(* IEC 61131-3 sources: BLM_BACKGROUND/src/PROGRAM_FILES/FC (part 3) *)

		GENERAL_STATE#STATE_END:
			CURRENT_STATE:=GENERAL_STATE#STATE_INIT;

	END_CASE;
	OutputState:=CURRENT_STATE;
END_FUNCTION_BLOCK

/*****************************************************************************
 * CHECKS WHETHER THE PIPE IS PRESENT ON THE^AL AND IS READY FOR LOADING, IF *
 *          NEGATIVE IT SETS THE STATUS AND POSITION TO UNDEFINED.           *
 *           IT ALSO RESETS OUTPUTS THAT CONTROL HAZARDOUS DEVICES           *
 *****************************************************************************/

FUNCTION_BLOCK FB_ResetAL

  VAR_EXTERNAL
    i_sys_OPMODE                          : INT;
    i_sys_current_prog	                  :INT;
    i_sys_AL_Robot                        :BOOL;
    OAddress                              : ARRAY [0..MAXDIGITALOUTPUT] OF Digital_Output;
    Disp                                  :ARRAY[(FIRST_DEVICE)..(FIRST_DEVICE+_MAXDEVICES#MAXDEVICES-1)] OF Device;
  END_VAR

  VAR_EXTERNAL CONSTANT
    AUTOMODE                              :INT;
    PROGRAM_JOG                      	    :SINT;
    TIPO_AL42                          	  :SINT;
    TIPO_AL42PLUS                      	  :SINT;
    MAXDIGITALOUTPUT                      :INT;
    OUT_ALZO_SOSTEGNO_TUBO_AL42           :INT;
    OUT_ABBASSO_SOSTEGNO_TUBO_AL42        :INT;
    CLAMP_CARGE                           :INT;
    FIRST_DEVICE                          :INT;
    AL42_STATO_CARICO                  	  :SINT;
    AT_STATE_UNDEFINED                	  :SINT;
    TIPO_AL5                          	  :SINT;
    TIPO_AL5_ROLAND                    	  :SINT;		//AL5 con sistema di misura ROLAND
    TIPO_AL5_LUNGO                    	  :SINT;
    AL5_CARICO_MACCHINA                	  :SINT;	//AL con tubo pronto in posizione di
                                                                //carico tubo in macchina con pinze
                                                                //chiuse, se presente traslatore avanti
    TIPO_AL5_BUNDLE                    	:SINT;
    TIPO_AL5_ROLAND_BUNDLE            	:SINT;		//AL5+BUNDLE con sistema di misura ROLAND
    TIPO_AL5_LUNGO_BUNDLE              	:SINT;	//AL5 speciale lungo 6mt+BUNDLE con sistema di misura ROLAND
    TIPO_MS0017                        	:SINT;	//Caricatore per ditta Sogefi
    TIPO_AL5_FUTABA                    	:SINT;	//Caricatore per ditta Futaba con ricerca saldatura Roland
    OUT_PRESSIONE_PNEUMATICA_AL         :INT;
  END_VAR

  VAR
    dwret     :DWORD;
    TipoAl    :SINT;
    dret      :DINT;
    Address   :DINT;
    StatoAsse :LREAL;
    Programma :INT;

		CURRENT_STATE:INT:=GENERAL_STATE#STATE_INIT;
		AL5_Sollevatore	:FB_AL5_Sollevatore;
		AL5Catene				:FB_AL5Catene;
  END_VAR
	VAR_OUTPUT
		OutputState:INT;
	END_VAR
	CASE CURRENT_STATE OF
		GENERAL_STATE#STATE_INIT:
			IF i_sys_OpMode=AUTOMODE THEN
				Programma:=I_SYS_Current_Prog;
			ELSE
				Programma:=PROGRAM_JOG;
			END_IF;
			// {#ifdef AL_BLM}
				i_sys_AL_Robot:=FALSE;
    		TipoAl:=IndicaTipoAl();
				CASE TipoAL OF
					TIPO_AL42, TIPO_AL42PLUS:
						//Abilitazione forzatura uscite
						oaddress[OUT_ALZO_SOSTEGNO_TUBO_AL42].enable_forzatura:=FALSE;
						oaddress[OUT_ABBASSO_SOSTEGNO_TUBO_AL42].enable_forzatura:=FALSE;
						(*dwret:=_resetTaskId(_task.motiontask_AL);*)
						Disp[CLAMP_CARGE].in_movimento:=FALSE;
						IF TestALReady()=TRUE THEN
							ImpostaAL(Stato:=AL42_STATO_CARICO, Movimento:=FALSE);
						ELSE
							//Stato CARICO AL42 non compatibile con la situazione reale dei
							//dispositivi quindi si mette ad indefinito lo stato del sistema
							Disp[CLAMP_CARGE].stato:=AT_STATE_UNDEFINED;
							Disp[CLAMP_CARGE].position:=AT_STATE_UNDEFINED;
						END_IF;
						CURRENT_STATE:=_FB_ResetAL#STATE_RESET_AL_RESET_USCITE_CARICO;

					TIPO_AL5, TIPO_AL5_ROLAND, TIPO_AL5_LUNGO:
						oaddress[OUT_ALZO_SOSTEGNO_TUBO_AL42].enable_forzatura:=FALSE;
						oaddress[OUT_ABBASSO_SOSTEGNO_TUBO_AL42].enable_forzatura:=FALSE;
						(*dwret:=_resetTaskId(_task.motiontask_AL);*)
						Disp[CLAMP_CARGE].in_movimento:=FALSE;
						IF TestALReady()=TRUE THEN
							ImpostaAL(Stato:=AL5_CARICO_MACCHINA, Movimento:=FALSE);
						ELSE
							//Stato CARICO AL42 non compatibile con la situazione reale dei
							//dispositivi quindi si mette ad indefinito lo stato del sistema
							Disp[CLAMP_CARGE].stato:=AT_STATE_UNDEFINED;
							Disp[CLAMP_CARGE].position:=AT_STATE_UNDEFINED;
						END_IF;
						CURRENT_STATE:=_FB_ResetAL#STATE_RESET_AL_RESET_USCITE_CARICO;

					TIPO_AL5_BUNDLE, TIPO_AL5_ROLAND_BUNDLE, TIPO_AL5_LUNGO_BUNDLE, TIPO_MS0017, TIPO_AL5_FUTABA:
						oaddress[OUT_ALZO_SOSTEGNO_TUBO_AL42].enable_forzatura:=FALSE;
						oaddress[OUT_ABBASSO_SOSTEGNO_TUBO_AL42].enable_forzatura:=FALSE;
						(*dwret:=_resetTaskId(_task.motiontask_AL);*)
						Disp[CLAMP_CARGE].in_movimento:=FALSE;
						IF TestALReady()=TRUE THEN
							ImpostaAL(Stato:=AL5_CARICO_MACCHINA, Movimento:=FALSE);
						ELSE
							//Stato CARICO AL42 non compatibile con la situazione reale dei
							//dispositivi quindi si mette ad indefinito lo stato del sistema
							Disp[CLAMP_CARGE].stato:=AT_STATE_UNDEFINED;
							Disp[CLAMP_CARGE].position:=AT_STATE_UNDEFINED;
						END_IF;
						CURRENT_STATE:=_FB_ResetAL#STATE_RESET_AL_AL5_SOLLEVATORE;

				ELSE
					//Per sicurezza abbasso la leva di carico, anche se teoricamente nell^AL42
					//non dovrebbe essere presente
					oaddress[OUT_PRESSIONE_PNEUMATICA_AL].stato:=TRUE;
					//Abilitazione forzatura uscite
					oaddress[OUT_ALZO_SOSTEGNO_TUBO_AL42].enable_forzatura:=TRUE;
					oaddress[OUT_ABBASSO_SOSTEGNO_TUBO_AL42].enable_forzatura:=TRUE;
					//Forzatura uscite per abbasso leva
					oaddress[OUT_ALZO_SOSTEGNO_TUBO_AL42].stato_forzatura:=FALSE;
					oaddress[OUT_ABBASSO_SOSTEGNO_TUBO_AL42].stato_forzatura:=TRUE;
					//Memorizzazione condizione di uscite per leva bassa per successivo reset
					//stato forzatura
					oaddress[OUT_ALZO_SOSTEGNO_TUBO_AL42].statopreforzatura:=SINT#0;
					oaddress[OUT_ABBASSO_SOSTEGNO_TUBO_AL42].statopreforzatura:=SINT#1;
					CURRENT_STATE:=_FB_ResetAL#STATE_RESET_AL_RESET_USCITE_CARICO;
				END_CASE;
			// {#endif} //FINE AL_BLM

    _FB_ResetAL#STATE_RESET_AL_AL5_SOLLEVATORE:
			// {#ifdef AL_BLM}
				AL5FrenoSollevatore(Stato:=FALSE);
				IF (AL5_Sollevatore.outputState<>GENERAL_STATE#STATE_END) THEN
					AL5_Sollevatore(Stato:=DEVICES_STATUS#ARRESTO, Attesa:=FALSE);
				ELSE
					AL5_Sollevatore(Stato:=DEVICES_STATUS#ARRESTO, Attesa:=FALSE);
					CURRENT_STATE:=_FB_ResetAL#STATE_RESET_AL_AL5_CATENE;
				END_IF;
			// {#endif} //FINE AL_BLM

    _FB_ResetAL#STATE_RESET_AL_AL5_CATENE:
			// {#ifdef AL_BLM}
				IF (AL5Catene.outputState<>GENERAL_STATE#STATE_END) THEN
					AL5Catene(Stato:=DEVICES_STATUS#ARRESTO);
				ELSE
					AL5Catene(Stato:=DEVICES_STATUS#ARRESTO);
					AL5LucePrenotazioneCarico(Stato:=FALSE);
					CURRENT_STATE:=_FB_ResetAL#STATE_RESET_AL_RESET_USCITE_CARICO;
				END_IF;
			// {#endif} //FINE AL_BLM

    _FB_ResetAL#STATE_RESET_AL_RESET_USCITE_CARICO:
			//Reset uscite dialogo AL con robot
			ALRobotProntoScarico(Stato:=FALSE, Programma:=Programma);
			ALRobotTuboLibero(Stato:=FALSE, Programma:=Programma);
			CURRENT_STATE:=GENERAL_STATE#STATE_END;

		GENERAL_STATE#STATE_END:
			CURRENT_STATE:=GENERAL_STATE#STATE_INIT;
	END_CASE;
	OutputState:=CURRENT_STATE;
END_FUNCTION_BLOCK

FUNCTION_BLOCK FB_ArrestaMotori
  VAR_INPUT
    Attesa  :BOOL;
  END_VAR
	VAR
		CURRENT_STATE	:INT:=GENERAL_STATE#STATE_INIT;
		// {#ifdef RUNNER} %%%%
		// 	TaglioRTL			:FB_TaglioRTL;
		// {#endif}
	END_VAR
	VAR_OUTPUT
		OutputState		:INT;
	END_VAR
	// CASE CURRENT_STATE OF %%%%
	// 	GENERAL_STATE#STATE_INIT:
  //   ;
	// 		// {#ifdef IPC_DISPOSITIVO} %%%%
	// 		// 	Set_Disp(Ndisp:=IPC_MOTORE, Stato:=RIPOSO, TimerRisparmio:=TRUE);
	// 		// {#endif}  //Fine IPC_DISPOSITIVO
	// 		// {#ifdef EFLEX_DH4010}
	// 		// 	Set_Disp(Ndisp:=SMUSSATORE_MOTORE, Stato:=RIPOSO, TimerRisparmio:=TRUE);
	// 		// {#endif}  //Fine EFLEX_DH4010
	// 		// {#ifdef RUNNER}
	// 		// 	Set_disp_position(Ndisp:=RULLATORE, Value:=RIPOSO, TimerRisparmio:=TRUE);
	// 		// 	WriteDigitalOutput(NumOutput:=OUT_MOTORE_FORATURA, Value:=FALSE);
	// 		// 	CURRENT_STATE:=STATE_ARRESTA_MOTORI_TAGLIORTL;
	// 		// {#else}
	// 		// 	CURRENT_STATE:=GENERAL_STATE#STATE_END;
	// 		// {#endif};  //Fine RUNNER

	// 	STATE_ARRESTA_MOTORI_TAGLIORTL:
	// 		{#ifdef RUNNER}
	// 			IF (TaglioRTL.outputState<>GENERAL_STATE#STATE_END) THEN
	// 				TaglioRTL(Velocita:=0, Attesa:=Attesa);
	// 			ELSE
	// 				TaglioRTL(Velocita:=0, Attesa:=Attesa);
	// 				CURRENT_STATE:=GENERAL_STATE#STATE_END;
	// 			END_IF;
	// 		{#endif};

	// 	GENERAL_STATE#STATE_END:
	// 		CURRENT_STATE:=GENERAL_STATE#STATE_INIT;

	// END_CASE;
	OutputState:=CURRENT_STATE;
END_FUNCTION_BLOCK

/**********************************************************************************************************
 *     ON 28/04/2014 ADDED CHAIN SYNCHRONISATION MANAGEMENT. WHEN ONE OF THE TWO LIMIT SWITCHES TO ON     *
 * WITH THE OTHER STILL AT OFF, ONLY THE CHAIN WITH THE SENSOR AT ON IS STOPPED. WHEN THE SENSOR THAT WAS *
 *    TO OFF ALSO SWITCHES TO ON, 0.1 IS ALLOWED TO ELAPSE WITH BOTH CHAINS STOPPED, AND THEN RESTARTS    *
 *                                              BOTH CHAINS                                               *
 **********************************************************************************************************/

// {#ifdef AL_BLM}
  FUNCTION_BLOCK FB_AL5Catene

    VAR_EXTERNAL
      TimerSistema                    :ARRAY[0..MAX_TIMER_SISTEMA-1] OF Timer;
    END_VAR

    VAR_EXTERNAL CONSTANT
      INP_AL5_SINCR_CATENA_SX                         :INT;
      T_SINCR_CATENE_AL5	                            :INT;
      MAX_TIMER_SISTEMA 	                            :USINT;
      INP_AL5_SINCR_CATENA_DX                         :INT;
    END_VAR

		VAR_INPUT
			Stato  :INT;
		END_VAR
		VAR
			dret  :DINT;

			CURRENT_STATE	:INT:=GENERAL_STATE#STATE_INIT;
			AL5CatenaDX		:FB_AL5CatenaDX;
			AL5CatenaSX		:FB_AL5CatenaSX;
			// {#ifdef MS0017}
			// 	AL5Catena3		:FB_AL5Catena3;
			// {#endif}
		END_VAR
		VAR_OUTPUT
			OutputState	:INT;
		END_VAR
		CASE CURRENT_STATE OF
				GENERAL_STATE#STATE_INIT:
					// {#ifdef MS0017} %%%%
					// 	CURRENT_STATE:=STATE_AL5_CATENE_MS0017_CATENA_DX;
					// {#else}
						IF Stato=DEVICES_STATUS#LAVORO THEN
							CURRENT_STATE:=_FB_AL5CATENE#STATE_AL5_CATENE_LAVORO;
						ELSE
							CURRENT_STATE:=_FB_AL5CATENE#STATE_AL5_CATENE_CATENA_DX_ALTRI_STATI;
						END_IF;
				// 	{#endif};

				// STATE_AL5_CATENE_MS0017_CATENA_DX:
				// 	{#ifdef MS0017}
				// 		IF (AL5CatenaDX.outputState<>GENERAL_STATE#STATE_END) THEN
				// 			AL5CatenaDX(Stato:=Stato);
				// 		ELSE
				// 			AL5CatenaDX(Stato:=Stato);
				// 			CURRENT_STATE:=STATE_AL5_CATENE_MS0017_CATENA_SX;
				// 		END_IF;
				// 	{#endif};

				// STATE_AL5_CATENE_MS0017_CATENA_SX:
				// 	{#ifdef MS0017}
				// 		IF (AL5CatenaSX.outputState<>GENERAL_STATE#STATE_END) THEN
				// 			AL5CatenaSX(Stato:=Stato);
				// 		ELSE
				// 			AL5CatenaSX(Stato:=Stato);
				// 			CURRENT_STATE:=STATE_AL5_CATENE_MS0017_CATENA_3;
				// 		END_IF;
				// 	{#endif};

				// STATE_AL5_CATENE_MS0017_CATENA_3:
				// 	{#ifdef MS0017}
				// 		IF (AL5Catena3.outputState<>GENERAL_STATE#STATE_END) THEN
				// 			AL5Catena3(Stato:=Stato);
				// 		ELSE
				// 			AL5Catena3(Stato:=Stato);
				// 			CURRENT_STATE:=GENERAL_STATE#STATE_END;
				// 		END_IF;
				// 	{#endif};

				_FB_AL5CATENE#STATE_AL5_CATENE_LAVORO:
					//Si sincronizza solo durante rotazione che porta il tubo verso le leve
					IF TestSincrCatene() THEN
						CURRENT_STATE:=_FB_AL5CATENE#STATE_AL5_CATENE_CATENA_DX_SINCRONIZZATE;
					ELSE
						CURRENT_STATE:=_FB_AL5CATENE#STATE_AL5_CATENE_NO_SINCRONIZZATE;
					END_IF;

        _FB_AL5CATENE#STATE_AL5_CATENE_CATENA_DX_SINCRONIZZATE:
					//Catene sincronizzate si comanda la rotazione
					IF (AL5CatenaDX.OutputState<>GENERAL_STATE#STATE_END) THEN
						AL5CatenaDX(Stato:=DEVICES_STATUS#LAVORO);
					ELSE
						AL5CatenaDX(Stato:=DEVICES_STATUS#LAVORO);
						CURRENT_STATE:=_FB_AL5CATENE#STATE_AL5_CATENE_CATENA_SX_SINCRONIZZATE;
					END_IF;

        _FB_AL5CATENE#STATE_AL5_CATENE_CATENA_SX_SINCRONIZZATE:
					//Catene sincronizzate si comanda la rotazione
					IF (AL5CatenaSX.OutputState<>GENERAL_STATE#STATE_END) THEN
						AL5CatenaSX(Stato:=DEVICES_STATUS#LAVORO);
					ELSE
						AL5CatenaSX(Stato:=DEVICES_STATUS#LAVORO);
						IF ReadDigitalInput(NumInput:=INP_AL5_SINCR_CATENA_SX, Verifica:=FALSE)=TRUE THEN
							//Se i due sensori sono a ON, si fa partire il timer che blocca la verifica della
							//sincronizzazione delle catene, così da evitare che durante la disattivazione dei sensori
							//si ricada in una nuova sincronizzazione. Attenzione che il tempo del timer deve
							//garantire la disattivazione dei finecorsa, ma essere più breve del tempo di rotazione
							//in modo che al successivo fronte di salita la sincronizzazione sia nuovamente abilitatata
							TimerSistema[T_SINCR_CATENE_AL5].Value:=1500;
            	TimerSistema[T_SINCR_CATENE_AL5].Status:=SINT#1;
						END_IF;
						CURRENT_STATE:=GENERAL_STATE#STATE_END;
					END_IF;

        _FB_AL5CATENE#STATE_AL5_CATENE_NO_SINCRONIZZATE:
					IF ReadDigitalInput(NumInput:=INP_AL5_SINCR_CATENA_SX, Verifica:=FALSE)=FALSE THEN
            //Occorre fermare la catena DX e ruotare la SX fino a quando si attiva il sensore SX
						CURRENT_STATE:=_FB_AL5CATENE#STATE_AL5_CATENE_NO_SYNC_CATENA_DX_ARRESTO;
					ELSE
						CURRENT_STATE:=_FB_AL5CATENE#STATE_AL5_CATENE_NO_SYNC_CATENA_SX_ARRESTO;
					END_IF;

        _FB_AL5CATENE#STATE_AL5_CATENE_NO_SYNC_CATENA_DX_ARRESTO:
					IF (AL5CatenaDX.OutputState<>GENERAL_STATE#STATE_END) THEN
						AL5CatenaDX(Stato:=DEVICES_STATUS#ARRESTO);
					ELSE
						AL5CatenaDX(Stato:=DEVICES_STATUS#ARRESTO);
						CURRENT_STATE:=_FB_AL5CATENE#STATE_AL5_CATENE_NO_SYNC_CATENA_SX_LAVORO_ATTESA_SYNC;
					END_IF;

        _FB_AL5CATENE#STATE_AL5_CATENE_NO_SYNC_CATENA_SX_LAVORO_ATTESA_SYNC:
					IF (AL5CatenaSX.OutputState<>GENERAL_STATE#STATE_END) THEN
						AL5CatenaSX(Stato:=DEVICES_STATUS#LAVORO);
					ELSE
						AL5CatenaSX(Stato:=DEVICES_STATUS#LAVORO);
						IF ReadDigitalInput(NumInput:=INP_AL5_SINCR_CATENA_SX, Verifica:=FALSE)=TRUE THEN
							CURRENT_STATE:=_FB_AL5CATENE#STATE_AL5_CATENE_NO_SYNC_CATENA_SX_ARRESTO_SYNC;
						END_IF;
					END_IF;

        _FB_AL5CATENE#STATE_AL5_CATENE_NO_SYNC_CATENA_SX_ARRESTO_SYNC:
					IF (AL5CatenaSX.OutputState<>GENERAL_STATE#STATE_END) THEN
						AL5CatenaSX(Stato:=DEVICES_STATUS#ARRESTO);
					ELSE
						AL5CatenaSX(Stato:=DEVICES_STATUS#ARRESTO);
						CURRENT_STATE:=_FB_AL5CATENE#STATE_AL5_CATENE_MANTIENI_CATENE_FERME;
					END_IF;

        _FB_AL5CATENE#STATE_AL5_CATENE_NO_SYNC_CATENA_SX_ARRESTO:
					IF (AL5CatenaSX.OutputState<>GENERAL_STATE#STATE_END) THEN
						AL5CatenaSX(Stato:=DEVICES_STATUS#ARRESTO);
					ELSE
						AL5CatenaSX(Stato:=DEVICES_STATUS#ARRESTO);
						CURRENT_STATE:=_FB_AL5CATENE#STATE_AL5_CATENE_NO_SYNC_CATENA_DX_LAVORO_ATTESA_SYNC;
					END_IF;

        _FB_AL5CATENE#STATE_AL5_CATENE_NO_SYNC_CATENA_DX_LAVORO_ATTESA_SYNC:
					IF (AL5CatenaDX.OutputState<>GENERAL_STATE#STATE_END) THEN
						AL5CatenaDX(Stato:=DEVICES_STATUS#LAVORO);
					ELSE
						AL5CatenaDX(Stato:=DEVICES_STATUS#LAVORO);
						IF ReadDigitalInput(NumInput:=INP_AL5_SINCR_CATENA_DX, Verifica:=FALSE)=TRUE THEN
							CURRENT_STATE:=_FB_AL5CATENE#STATE_AL5_CATENE_NO_SYNC_CATENA_DX_ARRESTO_SYNC;
						END_IF;
					END_IF;

        _FB_AL5CATENE#STATE_AL5_CATENE_NO_SYNC_CATENA_DX_ARRESTO_SYNC:
					IF (AL5CatenaDX.OutputState<>GENERAL_STATE#STATE_END) THEN
						AL5CatenaDX(Stato:=DEVICES_STATUS#ARRESTO);
					ELSE
						AL5CatenaDX(Stato:=DEVICES_STATUS#ARRESTO);
						CURRENT_STATE:=_FB_AL5CATENE#STATE_AL5_CATENE_MANTIENI_CATENE_FERME;
					END_IF;

        _FB_AL5CATENE#STATE_AL5_CATENE_MANTIENI_CATENE_FERME:
          //Mantenimento catene ferme, in pratica migliora la precisione della sincronizzazione
          //dret:=_waitTime(T#100ms);
					IF (AL5CatenaDX.OutputState<>GENERAL_STATE#STATE_END) THEN
						AL5CatenaDX(Stato:=DEVICES_STATUS#LAVORO);
					ELSE
						AL5CatenaDX(Stato:=DEVICES_STATUS#LAVORO);
						CURRENT_STATE:=_FB_AL5CATENE#STATE_AL5_CATENE_CATENA_SX_LAVORO_POST_SYNC;
					END_IF;

        _FB_AL5CATENE#STATE_AL5_CATENE_CATENA_SX_LAVORO_POST_SYNC:
					IF (AL5CatenaSX.OutputState<>GENERAL_STATE#STATE_END) THEN
						AL5CatenaSX(Stato:=DEVICES_STATUS#LAVORO);
					ELSE
						AL5CatenaSX(Stato:=DEVICES_STATUS#LAVORO);
						//Avvio del timer per bloccare la verifica di sincronizzazione durante la disattivazione
						//dei finecorsa
						TimerSistema[T_SINCR_CATENE_AL5].Value:=1000;
						TimerSistema[T_SINCR_CATENE_AL5].Status:=SINT#1;
						CURRENT_STATE:=GENERAL_STATE#STATE_END;
					END_IF;

        _FB_AL5CATENE#STATE_AL5_CATENE_CATENA_DX_ALTRI_STATI:
					IF (AL5CatenaDX.OutputState<>GENERAL_STATE#STATE_END) THEN
						AL5CatenaDX(Stato:=Stato);
					ELSE
						AL5CatenaDX(Stato:=Stato);
						CURRENT_STATE:=_FB_AL5CATENE#STATE_AL5_CATENE_CATENA_SX_ALTRI_STATI;
					END_IF;

        _FB_AL5CATENE#STATE_AL5_CATENE_CATENA_SX_ALTRI_STATI:
					IF (AL5CatenaSX.OutputState<>GENERAL_STATE#STATE_END) THEN
						AL5CatenaSX(Stato:=Stato);
					ELSE
						AL5CatenaSX(Stato:=Stato);
						CURRENT_STATE:=GENERAL_STATE#STATE_END;
					END_IF;

				GENERAL_STATE#STATE_END:
					CURRENT_STATE:=GENERAL_STATE#STATE_INIT;

		END_CASE;
		OutputState:=CURRENT_STATE;
	END_FUNCTION_BLOCK
// {#endif}  //Fine AL_BLM

/********************************************************
 * MANAGES THE JOG OF A REAL AXIS WITH ABSOLUTE ENCODER *
 ********************************************************/

FUNCTION_BLOCK FB_Homing_absolute

  VAR_EXTERNAL
    Axes                            :ARRAY[_FIRST_AXIS#FIRST_AXIS.._FIRST_AXIS#FIRST_AXIS+_CONST_VAR_DEF._MAXIS#MAXAXIS-1] OF ax;
    pm                              : ARRAY[_FIRST_AXIS#FIRST_AXIS.._FIRST_AXIS#FIRST_AXIS+_CONST_VAR_DEF._MAXIS#MAXAXIS-1] OF AxisParameters;
    cfg                             :_TYPE.Config_Struct;
    i_sys_AutoSetting					      :INT;
    i_sys_OPMODE                    : INT;
    i_sys_activedevice              : INT;
    Start_read								      : BOOL;
    mcHome									        :ARRAY[_FIRST_AXIS#FIRST_AXIS.._FIRST_AXIS#FIRST_AXIS+_CONST_VAR_DEF._MAXIS#MAXAXIS-1] OF MC_Home;
    UsoPLCOpen						          :BOOL;
  END_VAR

  VAR_EXTERNAL CONSTANT
    INACTIVE_DEACTIVATABLE_AXIS           :SINT;
    X1 :INT;
    REFMODE                               :INT;
    UNDEF_DEVICE                       	  :INT;
    SALVA_DATI_SIMOTION                   :SINT;
    driveObjectIdConstant                 : UINT;
        hardwareIdConstant                :WORD;
  END_VAR

  VAR_INPUT
    Asse      :INT;
    Position    :LREAL;
  END_VAR

  VAR
    PosAx     : REF_TO TO_SynchronousAxis;
    iret      :INT;
    dwret     :DWORD;
    dret      :DINT;

		CURRENT_STATE				:INT:=GENERAL_STATE#STATE_INIT;
		LetturaSinamicsREAL	: _READ_PARAMETER_SINGLE;
		ResetAxisBLM				:FB_ResetAxisBLM;
    Homing              : Homing;
  END_VAR

	VAR_OUTPUT
		OutputState	:INT;
		ReturnValue	:DINT;
	END_VAR

	CASE CURRENT_STATE OF
		GENERAL_STATE#STATE_INIT:
			IF pm[Asse].ma_stato_index=0 THEN
        PosAx:= AsSynchronousAxisRef(Axes[Asse].PosAx);
				IF pm[Asse].ma_asse_installato=INACTIVE_DEACTIVATABLE_AXIS AND PosAx^.Simulation.Mode=UDINT#1 THEN
					//Per gli assi in simulazione e disattivati da VGP3D, quindi con attivo il secondo encoder
					//ANALOG per fare in modo di non perdere la quota di index, occorre eliminare la simulazione
					//prima di fare l^index e poi ripristinarla
					IF (ResetAxisBLM.OutputState<>GENERAL_STATE#STATE_END) THEN
						ResetAxisBLM(Asse, TRUE);
					ELSE
						ResetAxisBLM(Asse, TRUE);
						CURRENT_STATE:=_FB_Homing_Absolute#STATE_HOMING_ABSOLUTE_HOME_SIMULATED_AXIS;
					END_IF;
				ELSE
					CURRENT_STATE:=_FB_Homing_Absolute#STATE_HOMING_ABSOLUTE_HOME_ACTIVATED_AXIS;
				END_IF;
			ELSE
				ReturnValue:=0;
				CURRENT_STATE:=GENERAL_STATE#STATE_END;
			END_IF;

    _FB_Homing_Absolute#STATE_HOMING_ABSOLUTE_HOME_SIMULATED_AXIS:
			Homing(Asse:=Asse, Quota:=Position, Modo:=EnumHomingMode#SET_OFFSET_OF_ABSOLUTE_ENCODER_BY_POSITION);
			// dret:=_enableAxisSimulation(axis:=Axes[Asse].PosAx, %%%%%
			// 														nextCommand:=IMMEDIATELY,
			// 														commandId:=_getCommandId());
			CURRENT_STATE:=GENERAL_STATE#STATE_END;

    _FB_Homing_Absolute#STATE_HOMING_ABSOLUTE_HOME_ACTIVATED_AXIS:
			Homing(Asse:=Asse, Quota:=Position, Modo:=EnumHomingMode#SET_OFFSET_OF_ABSOLUTE_ENCODER_BY_POSITION);
			IF (UsoPLCOpen) THEN
				CURRENT_STATE:=_FB_Homing_Absolute#STATE_HOMING_ABSOLUTE_WAIT_PLCOPEN_RESET;
			ELSE
				CURRENT_STATE:=_FB_Homing_Absolute#STATE_HOMING_ABSOLUTE_READ_NUMERO_SERIE_ENCODER;
			END_IF;

    _FB_Homing_Absolute#STATE_HOMING_ABSOLUTE_WAIT_PLCOPEN_RESET:
			IF (mcHome[Asse].done=TRUE) THEN
				CURRENT_STATE:=_FB_Homing_Absolute#STATE_HOMING_ABSOLUTE_READ_NUMERO_SERIE_ENCODER;
			END_IF;

    _FB_Homing_Absolute#STATE_HOMING_ABSOLUTE_READ_NUMERO_SERIE_ENCODER:
      posax:= AsSynchronousAxisRef(Axes[Asse].posax);
			IF posax^.VirtualAxis.Mode = UDINT#0 AND i_sys_OPMODE<>PI_COMMANDS_CODE#AUTOMODE AND Axes[Asse].IsSiemensAxis THEN

        IF NOT LetturaSinamicsREAL.Done THEN
          LetturaSinamicsREAL	(Start := Start_read,
                              driveObjectId      := driveObjectIdConstant,
                              hardwareId          := hardwareIdConstant,
                              parameterNumber     :=uint#463,
                              index              := uint#0);

				// IF (LetturaSinamicsREAL.outputState<>GENERAL_STATE#STATE_END) THEN
				// 	LetturaSinamicsREAL(log_address:=TO_DINT(Axes[Asse].PosAx.setconfigdata.TypeOfAxis.SetPointDriverInfo.logAddressIn),
				// 											par_number:=463,
				// 											sub_index:=0,
				// 											Verifica:=TRUE);
				ELSE
					Axes[Asse].NumSerieEncoder:=LetturaSinamicsREAL.Value_REAL;
                                LetturaSinamicsREAL	(Start := Start_read,
                                driveObjectId      := driveObjectIdConstant,
                                hardwareId          := hardwareIdConstant,
                                parameterNumber     :=uint#463,
                                index              := uint#0);
					// LetturaSinamicsREAL(log_address:=UDINT_TO_DINT(Assi[Asse].PosAx.setconfigdata.TypeOfAxis.SetPointDriverInfo.logAddressIn),
					// 										par_number:=463,
					// 										sub_index:=0,
					// 										Verifica:=TRUE);
          LetturaSinamicsREAL.Start :=false;
					CURRENT_STATE:=_FB_Homing_Absolute#STATE_HOMING_ABSOLUTE_SET_VALUES;
				END_IF;
			ELSE
				CURRENT_STATE:=_FB_Homing_Absolute#STATE_HOMING_ABSOLUTE_SET_VALUES;
			END_IF;

    _FB_Homing_Absolute#STATE_HOMING_ABSOLUTE_SET_VALUES:
			pm[Asse].MA_NUM_SERIE_ENCODER:=Axes[Asse].NumSerieEncoder;
      posax:= AsSynchronousAxisRef(Axes[Asse].posax);
			Axes[Asse].Homed:=PosAx^.StatusWord.%X5;
      PosAx^.PositionLimits_SW.Active:= TRUE;
			//Axes[Asse].PosAx.swlimit.state:=ACTIVE; ///???
			IF Asse=X1 THEN
				ImpostazioneOffsetX1(Offset:=cfg.OffsetMultiCannottoX1);
			END_IF;
			pm[Asse].ma_stato_index:=SINT#2;
			i_sys_AutoSetting:=SALVA_DATI_SIMOTION;
			(*dwret:=_startTaskId(_task.MotionTask_CambioConHard);*)
			IF i_sys_OPMODE=REFMODE THEN
				i_sys_activedevice:=UNDEF_DEVICE;
			END_IF;
			CURRENT_STATE:=GENERAL_STATE#STATE_END;

		GENERAL_STATE#STATE_END:
			CURRENT_STATE:=GENERAL_STATE#STATE_INIT;

	END_CASE;
	OutputState:=CURRENT_STATE;
END_FUNCTION_BLOCK

FUNCTION SistemaUtensili
  VAR
    Tasto1    :INT;
    Tasto2    :INT;
    Tasto3    :INT;
    Tasto4    :INT;
    i         :INT;
    Esito     :BOOL;
    Testa     :INT;
    EsitoDX,
    EsitoSX   :BOOL;
  END_VAR
  // {
  // #ifdef EFLEX_DH4010 %%%%
  // }
  //   BlmMxToolsTestine_1_5:=BlmMxToolsTestine_1_5_shadow;
  //   BlmMxToolsTestine_2_6:=BlmMxToolsTestine_2_6_shadow;
  // {
  // #else    //Fine EFLEX_DH4010
  // }
  //   BlmMxToolsOffPezzo:=BlmMxToolsOffPezzo_shadow;
  //   BlmMxCoppiaW3:=BlmMxCoppiaW3_shadow;
  //   BlmMxCoppiaW4:=BlmMxCoppiaW4_shadow;
  //   BlmMxCoppiaW5:=BlmMxCoppiaW5_shadow;
  //   BlmMxCoppiaW6:=BlmMxCoppiaW6_shadow;
  //   i_sys_Max_Ut_Macchina:=MaxTools_DX_Possibili+MaxTools_SX_Possibili;
	// 	BlmMxToolsDx:=BlmMxToolsDx_shadow;
	// 	BlmMxToolsSx:=BlmMxToolsSx_shadow;
  // {
  // #endif    //Fine NO EFLEX_DH4010
  // }
  // {
  // #ifdef SMART_SMART_A %%%%
  // }
  //   //Per poter eseguire il cambio raggio da una situazione di utensili tutti da una lato
  //   //e partenza della testa dal lato opposto, occore che anche la tabella relativa al lato
  //   //dove non ci sono utensili debba essere compilata con però la colonna QQt a 0
  //   IF MaxTools_DX_Installati=0 THEN
  //     //Tutti gli utensili installati sono sul lato SX ,si copia la tabella SX sulla DX
  //     //azzerando la colonna del raggio medio
  //     BLMMxToolsDX:=BLMMxToolsSX;
  //     FOR i:=1 TO MAXTOOLS*2 DO
  //       BLMMxToolsDX[i].qqt:=0;
  //     END_FOR;
  //   ELSE
  //     IF MaxTools_SX_Installati=0 THEN
  //       //Tutti gli utensili installati sono sul lato DX, si copia la tabella DX sulla SX
  //       //azzerando la colonna del raggio medio
  //       BLMMxToolsSX:=BLMMxToolsDX;
  //       FOR i:=1 TO MAXTOOLS*2 DO
  //         BLMMxToolsSX[i].qqt:=0;
  //       END_FOR;
  //     END_IF;
  //   END_IF;
  //   IF MaxTools_DX_Possibili=i_sys_Max_Ut_Macchina/2 THEN
  //     //Smart standard, metà utensili DX e metà utensili SX
  //     IF BlmMxToolsDx[1].Qqt>0.1 THEN
  //       Tasto1:=C_R_POSIZIONE_1;
  //     ELSE
  //       Tasto1:=C_R_POSIZIONE_1+MaxTools_DX_Possibili;
  //     END_IF;
  //     IF BlmMxToolsDx[2].Qqt>0.1 THEN
  //       Tasto2:=C_R_POSIZIONE_2;
  //     ELSE
  //       Tasto2:=C_R_POSIZIONE_2+MaxTools_DX_Possibili;
  //     END_IF;
  //     IF BlmMxToolsDx[3].Qqt>0.1 THEN
  //       Tasto3:=C_R_POSIZIONE_3;
  //     ELSE
  //       Tasto3:=C_R_POSIZIONE_3+MaxTools_DX_Possibili;
  //     END_IF;
  //     IF BlmMxToolsDx[4].Qqt>0.1 THEN
  //       Tasto4:=C_R_POSIZIONE_4;
  //     ELSE
  //       Tasto4:=C_R_POSIZIONE_4+MaxTools_DX_Possibili;
  //     END_IF;
  //   ELSE
  //     //Smart con solo utensili DX o SX
  //     Tasto1:=C_R_POSIZIONE_1;
  //     Tasto2:=C_R_POSIZIONE_2;
  //     Tasto3:=C_R_POSIZIONE_3;
  //     Tasto4:=C_R_POSIZIONE_4;
  //   END_IF;
  //   InizializzaKeyDisp(Tasto9:=Tasto1,
  //                      Tasto10:=Tasto2,
  //                      Tasto11:=Tasto3,
  //                      Tasto14:=Tasto4,
  //                      Tasto15:=-1,
  //                      Tasto16:=-1,
  //                      Tasto17:=-1,
  //                      Tasto18:=-1);
  // {
  // #endif	//Fine SMART_SMART_A
  // }
    // {
    // #ifdef ELECTMRL %%%%
    // }
		// 	IF BlmMxToolsDx[1].Qqt>0.1 THEN
		// 		Tasto1:=C_R_POSIZIONE_1;
		// 	ELSE
		// 		Tasto1:=C_R_POSIZIONE_1+MaxTools_DX_Possibili;
		// 	END_IF;
		// 	IF BlmMxToolsDx[2].Qqt>0.1 THEN
		// 		Tasto2:=C_R_POSIZIONE_2;
		// 	ELSE
		// 		Tasto2:=C_R_POSIZIONE_2+MaxTools_DX_Possibili;
		// 	END_IF;
		// 	IF BlmMxToolsDx[3].Qqt>0.1 THEN
		// 		Tasto3:=C_R_POSIZIONE_3;
		// 	ELSE
		// 		Tasto3:=C_R_POSIZIONE_3+MaxTools_DX_Possibili;
		// 	END_IF;
		// 	IF BlmMxToolsDx[4].Qqt>0.1 THEN
		// 		Tasto4:=C_R_POSIZIONE_4;
		// 	ELSE
		// 		Tasto4:=C_R_POSIZIONE_4+MaxTools_DX_Possibili;
		// 	END_IF;
		// 	InizializzaKeyDisp(Tasto9:=Tasto1,
		// 										 Tasto10:=Tasto2,
		// 										 Tasto11:=Tasto3,
		// 										 Tasto14:=Tasto4,
		// 										 Tasto15:=-1,
		// 										 Tasto16:=-1,
		// 										 Tasto17:=-1,
		// 										 Tasto18:=-1);
    // {
    // #endif //FINE ELECTMRL
    // }
  // {
  // #ifdef SMART_A %%%%
  // }
  //   //Imposta la zona dell^asse W4 all^interno della quale il sostegno tirante non
  //   //si può muovere
  //   ImpostaLimitiW4SostegnoTirante();
  // {
  // #endif	//Fine SMART_A
  // }
  //  {
  // #ifdef ETURN
  // }
  //   EsitoDX:=FALSE;
  //   EsitoSX:=FALSE;
  //   FOR i:=1 TO MAXTOOLS*2 DO
  //     IF BlmMxToolsDx[i].qqt>0.1 THEN
  //       Testa:=DX;
  //       EsitoDX:=TRUE;
  //       //Calcolo coordinate teoriche per P3 DX
  //       Esito:=ConvRealiTeoriciEturn(PosRealeQ:=BlmMxToolsDx[i].P3qq,
  //                                    PosRealeT:=BlmMxToolsDx[i].p3qt,
  //                                    LatoTesta:=Testa,
  //                                    PosTeoricaQ:=BlmMxToolsDx[i].p3qqt,
  //                                    PosTeoricaT:=BlmMxToolsDx[i].p3qtt);
  //       //Impostazione punto P4 per passaggio da Dx a Sx
  //       BlmMxToolsDx[i].p4qt:=BlmMxToolsDx[i].p3qt;
  //       BlmMxToolsDx[i].p4qq:=80;
  //       Esito:=ConvRealiTeoriciEturn(PosRealeQ:=BlmMxToolsDx[i].P4qq,
  //                                    PosRealeT:=BlmMxToolsDx[i].p4qt,
  //                                    LatoTesta:=Testa,
  //                                    PosTeoricaQ:=BlmMxToolsDx[i].p4qqt,
  //                                    PosTeoricaT:=BlmMxToolsDx[i].p4qtt);
  //       //Impostazione punto P5 (0, 90) per passaggio intermedio da Dx a Sx
  //       BlmMxToolsDx[i].p5qt:=0;
  //       BlmMxToolsDx[i].p5qq:=90;
  //       Esito:=ConvRealiTeoriciEturn(PosRealeQ:=BlmMxToolsDx[i].P5qq,
  //                                    PosRealeT:=BlmMxToolsDx[i].p5qt,
  //                                    LatoTesta:=Testa,
  //                                    PosTeoricaQ:=BlmMxToolsDx[i].p5qqt,
  //                                    PosTeoricaT:=BlmMxToolsDx[i].p5qtt);
  //     END_IF;
  //     IF BlmMxToolsSx[i].qqt>0.1 THEN
  //       Testa:=SX;
  //       EsitoSX:=TRUE;
  //       //Calcolo coordinate teoriche per P3 SX
  //       Esito:=ConvRealiTeoriciEturn(PosRealeQ:=BlmMxToolsSx[i].P3qq,
  //                                    PosRealeT:=BlmMxToolsSx[i].p3qt,
  //                                    LatoTesta:=Testa,
  //                                    PosTeoricaQ:=BlmMxToolsSx[i].p3qqt,
  //                                    PosTeoricaT:=BlmMxToolsSx[i].p3qtt);
  //       //Impostazione punto P4 per passaggio da Dx a Sx
  //       BlmMxToolsSx[i].p4qt:=BlmMxToolsSx[i].p3qt;
  //       BlmMxToolsSx[i].p4qq:=100;
  //       Esito:=ConvRealiTeoriciEturn(PosRealeQ:=BlmMxToolsSx[i].P4qq,
  //                                    PosRealeT:=BlmMxToolsSx[i].p4qt,
  //                                    LatoTesta:=Testa,
  //                                    PosTeoricaQ:=BlmMxToolsSx[i].p4qqt,
  //                                    PosTeoricaT:=BlmMxToolsSx[i].p4qtt);
  //       //Impostazione punto P5 (0, 90) per passaggio intermedio da Sx a Dx
  //       BlmMxToolsSx[i].p5qt:=0;
  //       BlmMxToolsSx[i].p5qq:=90;
  //       Esito:=ConvRealiTeoriciEturn(PosRealeQ:=BlmMxToolsSx[i].P5qq,
  //                                    PosRealeT:=BlmMxToolsSx[i].p5qt,
  //                                    LatoTesta:=Testa,
  //                                    PosTeoricaQ:=BlmMxToolsSx[i].p5qqt,
  //                                    PosTeoricaT:=BlmMxToolsSx[i].p5qtt);
  //     END_IF;
  //   END_FOR;
	// 	CalcolaUltimoUtPila();
  //   IF EsitoDX=TRUE AND EsitoSX=FALSE THEN
  //     //Significa che non è dichiarato nessun utensile sul lato SX, ma per poter fare il
  //     //rientro fuori ingombri mi servono le informazioni anche del lato SX, così imposto
  //     //un utensile fittizzio SX uguale a quello DX
  //     BlmMxToolsSX[1].qqt:=BlmMxToolsDX[i_sys_ultimo_ut_DX].qqt;
  //     BlmMxToolsSX[1].qtt:=BlmMxToolsDX[i_sys_ultimo_ut_DX].qtt;
  //     BlmMxToolsSX[1].qq:=180-BlmMxToolsDX[i_sys_ultimo_ut_DX].qq;
  //     BlmMxToolsSX[1].qt:=-BlmMxToolsDX[i_sys_ultimo_ut_DX].qt;
  //     BlmMxToolsSX[1].p2qqt:=BlmMxToolsDX[i_sys_ultimo_ut_DX].p2qqt;
  //     BlmMxToolsSX[1].p2qtt:=BlmMxToolsDX[i_sys_ultimo_ut_DX].p2qtt;
  //     BlmMxToolsSX[1].p2qq:=180-BlmMxToolsDX[i_sys_ultimo_ut_DX].p2qq;
  //     BlmMxToolsSX[1].p2qt:=-BlmMxToolsDX[i_sys_ultimo_ut_DX].p2qt;
  //     BlmMxToolsSX[1].p3qq:=180-BlmMxToolsDX[i_sys_ultimo_ut_DX].p3qq;
  //     BlmMxToolsSX[1].p3qt:=-BlmMxToolsDX[i_sys_ultimo_ut_DX].p3qt;
  //     BlmMxToolsSX[1].p3qqt:=BlmMxToolsDX[i_sys_ultimo_ut_DX].p3qqt;
  //     BlmMxToolsSX[1].p3qtt:=BlmMxToolsDX[i_sys_ultimo_ut_DX].p3qtt;
  //     BlmMxToolsSX[1].p4qq:=180-BlmMxToolsDX[i_sys_ultimo_ut_DX].p4qq;
  //     BlmMxToolsSX[1].p4qt:=-BlmMxToolsDX[i_sys_ultimo_ut_DX].p4qt;
  //     BlmMxToolsSX[1].p4qqt:=BlmMxToolsDX[i_sys_ultimo_ut_DX].p4qqt;
  //     BlmMxToolsSX[1].p4qtt:=BlmMxToolsDX[i_sys_ultimo_ut_DX].p4qtt;
  //     BlmMxToolsSX[1].p5qq:=180-BlmMxToolsDX[i_sys_ultimo_ut_DX].p5qq;
  //     BlmMxToolsSX[1].p5qt:=-BlmMxToolsDX[i_sys_ultimo_ut_DX].p5qt;
  //     BlmMxToolsSX[1].p5qqt:=BlmMxToolsDX[i_sys_ultimo_ut_DX].p5qqt;
  //     BlmMxToolsSX[1].p5qtt:=BlmMxToolsDX[i_sys_ultimo_ut_DX].p5qtt;
	// 		BlmMxToolsSx_shadow:=BlmMxToolsSx;
	// 		//Ricalcolo ultimo utensile pila sinistra doopo aver sistemato la BlmMxToolsSX
	// 		CalcolaUltimoUtPila();
  //   END_IF;
  //   IF EsitoSX=TRUE AND EsitoDX=FALSE THEN
  //     //Significa che non è dichiarato nessun utensile sul lato DX, ma per poter fare il
  //     //rientro fuori ingombri mi servono le informazioni anche del lato DX, così imposto
  //     //un utensile fittizzio DX uguale a quello SX
  //     BlmMxToolsDX[1].qqt:=BlmMxToolsSX[i_sys_ultimo_ut_SX].qqt;
  //     BlmMxToolsDX[1].qtt:=BlmMxToolsSX[i_sys_ultimo_ut_SX].qtt;
  //     BlmMxToolsDX[1].qq:=180-BlmMxToolsSX[i_sys_ultimo_ut_SX].qq;
  //     BlmMxToolsDX[1].qt:=-BlmMxToolsSX[i_sys_ultimo_ut_SX].qt;
  //     BlmMxToolsDX[1].p2qqt:=BlmMxToolsSX[i_sys_ultimo_ut_SX].p2qqt;
  //     BlmMxToolsDX[1].p2qtt:=BlmMxToolsSX[i_sys_ultimo_ut_SX].p2qtt;
  //     BlmMxToolsDX[1].p2qq:=180-BlmMxToolsSX[i_sys_ultimo_ut_SX].p2qq;
  //     BlmMxToolsDX[1].p2qt:=-BlmMxToolsSX[i_sys_ultimo_ut_SX].p2qt;
  //     BlmMxToolsDX[1].p3qq:=180-BlmMxToolsSX[i_sys_ultimo_ut_SX].p3qq;
  //     BlmMxToolsDX[1].p3qt:=-BlmMxToolsSX[i_sys_ultimo_ut_SX].p3qt;
  //     BlmMxToolsDX[1].p3qqt:=BlmMxToolsSX[i_sys_ultimo_ut_SX].p3qqt;
  //     BlmMxToolsDX[1].p3qtt:=BlmMxToolsSX[i_sys_ultimo_ut_SX].p3qtt;
  //     BlmMxToolsDX[1].p4qq:=180-BlmMxToolsSX[i_sys_ultimo_ut_SX].p4qq;
  //     BlmMxToolsDX[1].p4qt:=-BlmMxToolsSX[i_sys_ultimo_ut_SX].p4qt;
  //     BlmMxToolsDX[1].p4qqt:=BlmMxToolsSX[i_sys_ultimo_ut_SX].p4qqt;
  //     BlmMxToolsDX[1].p4qtt:=BlmMxToolsSX[i_sys_ultimo_ut_SX].p4qtt;
  //     BlmMxToolsDX[1].p5qq:=180-BlmMxToolsSX[i_sys_ultimo_ut_SX].p5qq;
  //     BlmMxToolsDX[1].p5qt:=-BlmMxToolsSX[i_sys_ultimo_ut_SX].p5qt;
  //     BlmMxToolsDX[1].p5qqt:=BlmMxToolsSX[i_sys_ultimo_ut_SX].p5qqt;
  //     BlmMxToolsDX[1].p5qtt:=BlmMxToolsSX[i_sys_ultimo_ut_SX].p5qtt;
	// 		BlmMxToolsDx_shadow:=BlmMxToolsDx;
	// 		CalcolaUltimoUtPila();
	// 		//Ricalcolo ultimo utensile pila destra doopo aver sistemato la BlmMxToolsDX
  //   END_IF;
	// 	//Copia anche nella shadow i dati calcolati perchè servono nella gestione delle piattine
	// 	BlmMxToolsDx_shadow:=BlmMxToolsDx;
	// 	BlmMxToolsSx_shadow:=BlmMxToolsSx;
  // {
  // #endif    //Fine ETURN
  // }
  ;
END_FUNCTION

/*********************************************
 * RESETS THE REQUIRED STATUS OF ALL DEVICES *
 *********************************************/

FUNCTION ResetStatoRichiesto

  VAR_EXTERNAL
    Disp                            :ARRAY[(FIRST_DEVICE)..(FIRST_DEVICE+_MAXDEVICES#MAXDEVICES-1)] OF Device;
  END_VAR

  VAR_EXTERNAL CONSTANT
    FIRST_DEVICE                    :INT;
  END_VAR

  VAR
    i  :INT;
  END_VAR
  FOR i:=FIRST_DEVICE TO FIRST_DEVICE+_MAXDEVICES#MAXDEVICES-1 DO
    disp[i].StatoRichiesto:=-1;
  END_FOR;
END_FUNCTION

FUNCTION ResetOutCaricoScaricoRobot

  VAR_EXTERNAL CONSTANT
    OUT_CARICO_MACCHINA_PRONTA                    :INT;
    OUT_CARICO_MACCHINA_PRONTA_DPCOUPLER          :INT;
    OUT_FCY                                       :INT;
    OUT_CARICO_MACCHINA_TUBO_PRESO                :INT;
    OUT_CARICO_MACCHINA_TUBO_PRESO_DPCOUPLER      :INT;
    OUT_SCARICO_MACCHINA_PRONTA                   :INT;
    OUT_SCARICO_MACCHINA_PRONTA_DPCOUPLER         :INT;
    OUT_SCARICO_MACCHINA_TUBO_LIBERO			        :INT;
    OUT_SCARICO_MACCHINA_TUBO_LIBERO_DPCOUPLER      :INT;
    OUT_CODIFICA_PROGRAMMA_OK_DPCOUPLER             :INT;
  END_VAR
  // {
  // #ifdef CARICO_AUTOMATICO
  // }
    WriteDigitalOutput(NumOutput:=OUT_CARICO_MACCHINA_PRONTA, Value:=FALSE, Verifica:=FALSE);
    WriteDigitalOutput(NumOutput:=OUT_CARICO_MACCHINA_PRONTA_DPCOUPLER, Value:=FALSE, Verifica:=FALSE);
    WriteDigitalOutput(NumOutput:=OUT_FCY, Value:=FALSE, Verifica:=FALSE);
    WriteDigitalOutput(NumOutput:=OUT_CARICO_MACCHINA_TUBO_PRESO, Value:=FALSE, Verifica:=FALSE);
    WriteDigitalOutput(NumOutput:=OUT_CARICO_MACCHINA_TUBO_PRESO_DPCOUPLER, Value:=FALSE, Verifica:=FALSE);
    // {
    // #ifndef DH4010 %%%%
    // }
    //   WriteDigitalOutput(NumOutput:=OUT_CARICO_MACCHINA_X1_FI, Value:=FALSE, Verifica:=FALSE);
    //   WriteDigitalOutput(NumOutput:=OUT_CARICO_MACCHINA_X1_FI_DPCOUPLER, Value:=FALSE, Verifica:=FALSE);
    //   WriteDigitalOutput(NumOutput:=OUT_CARICO_TUBO_PRESENTE_AL, Value:=FALSE, Verifica:=FALSE);
    //   WriteDigitalOutput(NumOutput:=OUT_CARICO_TUBO_PRESENTE_AL_DPCOUPLER, Value:=FALSE, Verifica:=FALSE);
    //   WriteDigitalOutput(NumOutput:=OUT_CARICO_TUBO_LIBERO_AL, Value:=FALSE, Verifica:=FALSE);
    //   WriteDigitalOutput(NumOutput:=OUT_CARICO_TUBO_LIBERO_AL_DPCOUPLER, Value:=FALSE, Verifica:=FALSE);
    //   WriteDigitalOutput(NumOutput:=OUT_CARICO_TUBO_KO_AL_DPCOUPLER, Value:=FALSE, Verifica:=FALSE);
		// {
    // #endif  //Fine DH4010
    // }
  // {
  // #endif  //Fine CARICO_AUTOMATICO
  // }
  WriteDigitalOutput(NumOutput:=OUT_SCARICO_MACCHINA_PRONTA, Value:=FALSE, Verifica:=FALSE);
  WriteDigitalOutput(NumOutput:=OUT_SCARICO_MACCHINA_PRONTA_DPCOUPLER, Value:=FALSE, Verifica:=FALSE);
  WriteDigitalOutput(NumOutput:=OUT_SCARICO_MACCHINA_TUBO_LIBERO, Value:=FALSE, Verifica:=FALSE);
  WriteDigitalOutput(NumOutput:=OUT_SCARICO_MACCHINA_TUBO_LIBERO_DPCOUPLER, Value:=FALSE, Verifica:=FALSE);
  WriteDigitalOutput(NumOutput:=OUT_CODIFICA_PROGRAMMA_OK_DPCOUPLER, Value:=FALSE, Verifica:=FALSE);
	ResetCodificaPezzo();
END_FUNCTION

FUNCTION OutScartoLavorazione
  VAR_INPUT
    Stato  :BOOL;
  END_VAR
  // {
  // #ifndef ORBITALE %%%%
  // }
  //   IF cfg.TipoTaglioColtello=TAGLIO_COLTELLO_PRIMA_VER THEN
  //     //Prima versione taglio a coltello, la temporizzazione avviene mediante un timer elettromeccanico
  //     WriteDigitalOutput(NumOutput:=OUT_ESPULSIONE_SCARTO_LAVORAZIONE, Value:=Stato);
  //   ELSE
  //     //Seconda versione taglio a coltello, la temporizzazione è software
  //     IF Stato=TRUE THEN
  //       IF TimerSistema[T_SCARTO_LAVORAZ].Stato=0 THEN
  //         TimerSistema[T_SCARTO_LAVORAZ].Value:=(TempoSoffioSfridiTaglioColtello*1000)+VALORE_FINE_TIMER;
  //         TimerSistema[T_SCARTO_LAVORAZ].Stato:=1;
  //       END_IF;
  //     END_IF;
  //   END_IF;
  // {
  // #endif  //Fine NO ORBITALE
  // }
  ;
END_FUNCTION

FUNCTION MacchinaInWarning

  VAR_EXTERNAL
    i_sys_DpCoupler                 :BOOL;
    i_sys_PnCoupler                 :BOOL;
  END_VAR

  VAR_EXTERNAL CONSTANT
    MAXDIGITALOUTPUT                    :INT;
    OUT_MACCHINA_IN_WARNING_DPCOUPLER               :INT;
  END_VAR

  VAR_INPUT
    Stato  :BOOL;
  END_VAR

  IF i_sys_DpCoupler=TRUE OR i_sys_PnCoupler=TRUE THEN
		WriteDigitalOutput(NumOutput:=OUT_MACCHINA_IN_WARNING_DPCOUPLER, Value:=Stato);
	ELSE
		WriteDigitalOutput(NumOutput:=OUT_MACCHINA_IN_WARNING_DPCOUPLER, Value:=FALSE);
  END_IF;
END_FUNCTION

/******************************************************************
 * RESET STRUCTURE STATUS_OUT WHERE I STORE DIGITAL OUTPUT STATUS *
 ******************************************************************/
FUNCTION Res_StatoOut

  VAR_EXTERNAL
    Stato_Out                                 :ARRAY[0..MAXDIGITALOUTPUT] OF Struttura_Stato_Out;
  END_VAR

  VAR_EXTERNAL CONSTANT
    MAXDIGITALOUTPUT                    :INT;
  END_VAR
  VAR
    i:DINT;
  END_VAR
  FOR i:=0 TO MAXDIGITALOUTPUT DO
    Stato_Out[i].Stato:=BOOL#0;
  END_FOR;
END_FUNCTION

FUNCTION ImpostaOutWeld
  VAR_INPUT
    Stato  :BOOL;
  END_VAR
  // {
  // #ifndef ORBITALE
  // }
  //   WriteDigitalOutput(NumOutput:=OUT_WELD, Value:=Stato);
  // {
  // #endif  //Fine NO ORBITALE
  // }
  ;
END_FUNCTION

FUNCTION ImpostaOutMisuraAnima
  VAR_INPUT
    Stato  :BOOL;
  END_VAR
  // {
  // #ifndef ORBITALE
  // }
  //   WriteDigitalOutput(NumOutput:=OUT_MISURA_ANIMA_KO, Value:=Stato);
  // {
  // #endif  //Fine NO ORBITALE
  // }
  ;
END_FUNCTION

FUNCTION Set_Disp_Position

  VAR_EXTERNAL
      Disp                            :ARRAY[(FIRST_DEVICE)..(FIRST_DEVICE+_MAXDEVICES#MAXDEVICES-1)] OF Device;
  END_VAR

    VAR_EXTERNAL CONSTANT
      FIRST_DEVICE                    :INT;
      DISP_IN_V_C                     :SINT;
      DISP_IN_V                       :SINT;
      RIPOSO                          :SINT;
  END_VAR

  VAR_INPUT
    Ndisp						:INT;
    Value						:LREAL;
    TimerRisparmio	:BOOL;
  END_VAR
  VAR
    Valore          :REAL;
  END_VAR

  IF Disp[NDisp].enable THEN
    Disp[NDisp].statorichiesto:=TO_REAL(Value);
    CASE Disp[Ndisp].tipoin OF
      DISP_IN_V:
        Set_Disp(Ndisp:=Ndisp, Stato:=TO_INT(Value), TimerRisparmio:=TimerRisparmio);
      DISP_IN_V_C:
        Valore:=TO_REAL(Value);
        // IF _getStateOfTaskId(_task.motiontask_AUTO)<>TASK_STATE_STOPPED THEN
        //   SetDispComplesso(NDisp:=NDisp, Value:=Valore, Attesa:=TRUE, TimerRisparmio:=TimerRisparmio);
        // ELSE
          //Se non è attivo AUTOMODE non si esegue attesa, altrimenti si
          //superano i tempi del background
          SetDispComplesso(NDisp:=NDisp, Value:=Valore, Attesa:=FALSE, TimerRisparmio:=TimerRisparmio);
        // END_IF;
    ELSE
      //Dispositivo reale si accettano due stati possibili LAVORO o RIPOSO
      IF Value>(DISP[Ndisp].Limite_Lavoro-DISP[Ndisp].Limite_Riposo)/2 THEN
        Set_Disp(Ndisp:=Ndisp, Stato:=DEVICES_STATUS#LAVORO, TimerRisparmio:=TimerRisparmio);
      ELSE
        Set_Disp(Ndisp:=Ndisp, Stato:=RIPOSO, TimerRisparmio:=TimerRisparmio);
      END_IF;
    END_CASE;
  END_IF;
END_FUNCTION

FUNCTION ComandaRadar

    VAR_EXTERNAL CONSTANT
      AUTOMODE                              :INT;
      MIN_ZONA_RADAR_VGP                    :SINT;
    END_VAR

    VAR_EXTERNAL
      Programmi                      :ARRAY[0.._CONST_VAR_DEF._MPROGRAMS#MAXPROGRAMS - UINT#1] OF Programma;
    END_VAR

  VAR_INPUT
		Programma			:DINT;
		ModoOperativo	:INT;
  END_VAR
  // {
  // #ifndef PROFINET
  // }
    IF ModoOperativo=AUTOMODE THEN
      IF Programmi[Programma].UsoRadar_Pezzo>MIN_ZONA_RADAR_VGP THEN
        AttivaProgrammaRadar(Codice:=Programmi[Programma].UsoRadar_Pezzo);
      END_IF;
    ELSE
      IF Programmi[Programma].usoradar_manuale>MIN_ZONA_RADAR_VGP THEN
        AttivaProgrammaRadar(Codice:=Programmi[Programma].usoradar_manuale);
      END_IF;
    END_IF;
  // {
  // #endif  //Fine NO PROFINET
  // }
  ;
END_FUNCTION

/**************************************************
 * SET THE OUTPUT THAT ACTIVATES THE CARM7 PUMPER *
 **************************************************/

FUNCTION PompatoreCARM7
  VAR_INPUT
    Stato  :BOOL;
  END_VAR
  ;
  // {
  // #ifdef SMART %%%%
  // }
  //   IF disp[CLAMP_CARGE].enable=TRUE THEN
  //     WriteDigitalOutput(NumOutput:=OUT_CARICO_RIC_CAR, Value:=Stato);
  //   END_IF;
  // {
  // #endif    //Fine SMART
  // }
END_FUNCTION

/*********************************************************************************
 * THE FUNCTION TAKES CARE OF SETTING THE JOB STATUS FOR PROTUBE AND WEBAPP DATA *
 *          THE STATUS SUSPENDED CAN^ ONLY BE SET FOLLOWING A TRANSFER           *
 *                             OF A NEW JOBID BY VGP                             *
 *********************************************************************************/

FUNCTION SetJobState

  VAR_EXTERNAL
    ProTube                         :Produzione;
    i_sys_ModoPezzoSeguente         : INT;
    WebApp                          :WebApplication;
  END_VAR

  VAR_EXTERNAL CONSTANT
    MODO_PEZZO_SEGUENTE                             :SINT;
    MODO_PEZZO_STANDARD                     :SINT;
  END_VAR

	VAR_INPUT
		Stato						:INT;
		ForzaturaStato	:BOOL:=FALSE;
		DatiProTube			:BOOL:=TRUE;
		DatiWebApp			:BOOL:=TRUE;
	END_VAR

	IF Protube.jobid=J_ID_RESET#JOB_ID_RESET AND Protube.JobGUID='' AND i_sys_modopezzoseguente>MODO_PEZZO_STANDARD THEN
		//Protube.jobstate:=JOB_STATE_NULLO;
		;
	ELSE
		IF DatiProTube=TRUE THEN
			IF i_sys_modopezzoseguente>=MODO_PEZZO_SEGUENTE OR ForzaturaStato=TRUE THEN
				Protube.jobstate:=Stato;
			END_IF;
		END_IF;
	END_IF;
	IF DatiWebApp=TRUE THEN
		IF WebApp.wd_job_code<>'-1' THEN
			WebApp.wd_job_state:=Stato;
		ELSE
			//WebApp.wd_job_state:=JOB_STATE_NULLO;
			;
		END_IF;
	END_IF;
END_FUNCTION

FUNCTION ImpostaAL

  VAR_EXTERNAL
    Disp                                 :ARRAY[(FIRST_DEVICE)..(FIRST_DEVICE+_MAXDEVICES#MAXDEVICES-1)] OF Device;
    Programmi                            :ARRAY[0.._CONST_VAR_DEF._MPROGRAMS#MAXPROGRAMS - UINT#1] OF Programma;
    i_sys_current_prog	                 :INT;
    AL_LunghezzaTubo                     :LREAL;
  END_VAR

  VAR_EXTERNAL CONSTANT
    FIRST_DEVICE                    :INT;
    AL42_STATO_CARICO               :SINT;
    AL5_CARICO_MACCHINA             :SINT;
    CLAMP_CARGE                     :INT;
    AL42PLUS_STATO_CARICO           :SINT;
  END_VAR

  VAR_INPUT
    Stato    :INT;
    Movimento  :BOOL;
  END_VAR
  // {
  // #ifdef AL_BLM
  // }
    Disp[CLAMP_CARGE].in_movimento:=Movimento;
    Disp[CLAMP_CARGE].stato:=Stato;
    Disp[CLAMP_CARGE].position:=Stato;
    IF Stato=AL42_STATO_CARICO OR
       Stato=AL42PLUS_STATO_CARICO OR
       Stato=AL5_CARICO_MACCHINA THEN
      //Al momento dell^impostazione dello stato carico si memorizza la lunghezza
      //del tubo preso sull^AL
      AL_LunghezzaTubo:=Programmi[i_sys_current_prog].LunghezzaTuboEsecuzione;
    END_IF;
  // {
  // #endif  //Fine AL_BLM
  // }
  ;
END_FUNCTION

/**************************************************************************************************
 * RESETTING DISTANCE FROM THE END OF POSITIONING WITH POSSIBLE MAINTENANCE OF THE INDICATED AXIS *
 **************************************************************************************************/

FUNCTION AzzeramentoDistanceTogo

  VAR_EXTERNAL
    i_sys_PosFinale							:ARRAY[(_FIRST_AXIS#FIRST_AXIS) .. (_FIRST_AXIS#FIRST_AXIS+_MAXIS#MAXAXIS -1)] OF LREAL;
  END_VAR

  VAR_EXTERNAL CONSTANT
    MY_BIG_VALUE_INT                :INT;
    MY_BIG_VALUE_REAL               :REAL;
  END_VAR

  VAR_INPUT
    Asse  :INT:=-MY_BIG_VALUE_INT;
  END_VAR
  VAR
    i     :INT;
  END_VAR
  FOR i:=_FIRST_AXIS#FIRST_AXIS TO _FIRST_AXIS#FIRST_AXIS+_MAXIS#MAXAXIS-1 BY 1 DO
    IF Asse>=_FIRST_AXIS#FIRST_AXIS AND Asse<=_FIRST_AXIS#FIRST_AXIS+_MAXIS#MAXAXIS-1 THEN
      IF i<>Asse THEN
        i_sys_PosFinale[i]:=-MY_BIG_VALUE_REAL;
      END_IF;
    ELSE
      i_sys_PosFinale[i]:=-MY_BIG_VALUE_REAL;
    END_IF;
  END_FOR;
END_FUNCTION

FUNCTION_BLOCK FB_AL5_Sollevatore

  VAR_EXTERNAL CONSTANT
    AL5_SOLLEVATORE_FASCIO                        :INT;  //42
    OUT_AL5_ALZO_FASCIO                           :INT;
    OUT_AL5_ABBASSO_FASCIO                        :INT;
    TRC_AL5_SOLLEVATORE_FASCIO_ALTO               :INT;
    TRC_AL5_SOLLEVATORE_FASCIO_BASSO              :INT;
  END_VAR

  VAR_INPUT
    Stato    :INT;
    Attesa  :BOOL;
  END_VAR

  VAR
    dret    :DINT;

		CURRENT_STATE	:INT:=GENERAL_STATE#STATE_INIT;
		Wait_Disp			:FB_Wait_disp;
		VerificaStop	:FB_VerificaStop;
  END_VAR
	VAR_OUTPUT
		OutputState	:INT;
	END_VAR
  ;
  {
  #ifdef AL_BLM
  }
		CASE CURRENT_STATE OF
			GENERAL_STATE#STATE_INIT:
				IF STATO=DEVICES_STATUS#ARRESTO THEN
					AL5FrenoSollevatore(Stato:=FALSE);
					WriteDigitalOutput(NumOutput:=OUT_AL5_ALZO_FASCIO, Value:=FALSE);
					WriteDigitalOutput(NumOutput:=OUT_AL5_ABBASSO_FASCIO, Value:=FALSE);
					CURRENT_STATE:=GENERAL_STATE#STATE_END;
				ELSE
					IF (VerificaStop.OutputState<>GENERAL_STATE#STATE_END) THEN
						VerificaStop();
					ELSE
						VerificaStop();
						AL5FrenoSollevatore(Stato:=TRUE);
						Set_Disp(Ndisp:=AL5_SOLLEVATORE_FASCIO, Stato:=Stato, TimerRisparmio:=TRUE);
						IF Attesa=TRUE THEN
							CURRENT_STATE:=_FB_AL5_Sollevatore#STATE_SOLLEVATORE_WAIT_SOLLEVATORE;
						ELSE
							CURRENT_STATE:=_FB_AL5_Sollevatore#STATE_SOLLEVATORE_VERIFICA_STOP;
						END_IF;
					END_IF;
				END_IF;

        _FB_AL5_Sollevatore#STATE_SOLLEVATORE_WAIT_SOLLEVATORE:
				IF Stato=DEVICES_STATUS#LAVORO THEN
          set_trace(Code:=TRC_AL5_SOLLEVATORE_FASCIO_ALTO);
        ELSE
          set_trace(Code:=TRC_AL5_SOLLEVATORE_FASCIO_BASSO);
        END_IF;
				IF (wait_disp.outputstate<>GENERAL_STATE#STATE_END) THEN
					wait_disp(Device:=AL5_SOLLEVATORE_FASCIO, State:=Stato, Trace:=FALSE);
				ELSE
					reset_trace(Code:=TRC_AL5_SOLLEVATORE_FASCIO_ALTO);
        	reset_trace(Code:=TRC_AL5_SOLLEVATORE_FASCIO_BASSO);
					VerificaStop();
					CURRENT_STATE:=GENERAL_STATE#STATE_END;
				END_IF;

        _FB_AL5_Sollevatore#STATE_SOLLEVATORE_VERIFICA_STOP:
				IF (VerificaStop.OutputState<>GENERAL_STATE#STATE_END) THEN
					VerificaStop();
				ELSE
					VerificaStop();
					CURRENT_STATE:=GENERAL_STATE#STATE_END;
				END_IF;

			GENERAL_STATE#STATE_END:
				CURRENT_STATE:=GENERAL_STATE#STATE_INIT;
		END_CASE;
		OutputState:=CURRENT_STATE;
  // {
  // #endif  //Fine AL_BLM
  // }
END_FUNCTION_BLOCK

/*********************************
 * RETURNS THE TYPE OF ACTIVE AL *
 *********************************/

FUNCTION IndicaTipoAl:SINT

  VAR_EXTERNAL
    cfg                             :_TYPE.Config_Struct;
  END_VAR

  VAR_EXTERNAL CONSTANT
    TIPO_CARM                          	            :SINT;
  END_VAR
  // {
  // #ifdef AL_BLM
  // }
    IF cfg.i_sys_caricatoreblm_dx>=TIPO_CARM THEN
      IndicaTipoAl:=cfg.i_sys_caricatoreblm_dx;
    ELSE
      IF cfg.i_sys_caricatoreblm_sx>=TIPO_CARM THEN
        IndicaTipoAl:=cfg.i_sys_caricatoreblm_sx;
      ELSE
        IndicaTipoAl:=SINT#0;
      END_IF;
    END_IF;
  // {
  //   #else    //Fine AL_BLM
  // }
    IndicaTipoAl:=SINT#0;
  // {
  //   #endif    //Fine NO AL_BLM
  // }
END_FUNCTION

/*********************************************************************************
 * CHECK IF THE TUBE IS PRESENT ON THE^AL AND READY FOR LOADING INTO THE MACHINE *
 *********************************************************************************/

FUNCTION TestALReady:BOOL

  VAR_EXTERNAL CONSTANT
    PROGRAM_JOG                      	:SINT;
  END_VAR

  VAR_EXTERNAL
    i_sys_OPMODE                    : INT;
  END_VAR

  VAR
    ProgrammaAttivo                       :DINT;
    TipoAl                                :SINT;
    i_sys_current_prog	                  :INT;
  END_VAR

  TestALReady:=FALSE;
  TipoAl:=IndicaTipoAl();
  IF i_sys_OpMode=PI_COMMANDS_CODE#AUTOMODE THEN
    ProgrammaAttivo:=I_SYS_Current_Prog;
  ELSE
    ProgrammaAttivo:=PROGRAM_JOG ;
  END_IF;
  // {
  // #ifndef MS0017 %%%%
  // }
  //   CASE TipoAl OF
  //     TIPO_AL42:
  //       IF TestTuboAL42()=2 AND
  //          Disp[AL42SOSTEGNO].stato=RIPOSO AND
  //          (Disp[AL42SPINTORE].stato=DEVICES_STATUS#LAVORO OR i_sys_SenzaTubo=TRUE) THEN
  //         TestALReady:=TRUE;
  //       ELSE
  //         IF Disp[PINZA_CARICO].stato=AL42_STATO_CARICO THEN
  //           //Reset stato carico se la posizione dei dispositivi non
  //           //è compatibile
  //           Disp[PINZA_CARICO].stato:=AL_STATO_INDEFINITO;
  //         END_IF;
  //       END_IF;
  //     TIPO_AL42PLUS:
  //       //Condizioni per essere nello stato CARICO:
  //       //- Pinze chiuse
  //       //- Tubo presente in pinza
  //       //- Traslatore avanti
  //       //- L1 alla quota di carico
  //       IF readdigitalinput(NumInput:=INP_PRESENZA_PEZZO_SU_PINZA_AL42_PLUS)=FALSE AND
  //          i_sys_SenzaTubo=FALSE THEN
  //         TestALReady:=FALSE;
  //       ELSE
  //         IF readdigitalinput(NumInput:=INP_PINZE_CHIUSE_AL42_PLUS)=TRUE AND
  //            readdigitalinput(NumInput:=INP_PINZE_APERTE_AL42_PLUS)=FALSE AND
  //            readdigitalinput(NumInput:=INP_TRASLAZIONE_AVANTI_AL42_PLUS)=TRUE AND
  //            readdigitalinput(NumInput:=INP_TRASLAZIONE_INDIETRO_AL42_PLUS)=FALSE AND
  //            ABS(Axes[L1].PosAx.positioningState.actualPosition-Programmi[ProgrammaAttivo].DatiAL.L1PosCarico)<pm[L1].ma_standstill_pos_tol THEN
  //           TestALReady:=TRUE;
  //         END_IF;
  //       END_IF;
  //     TIPO_AL5, TIPO_AL5_BUNDLE, TIPO_AL5_ROLAND, TIPO_AL5_ROLAND_BUNDLE,
  //     TIPO_AL5_LUNGO, TIPO_AL5_LUNGO_BUNDLE, TIPO_AL5_FUTABA:
  //       //Condizioni per essere nello stato CARICO:
  //       //- Pinze non aperte
  //       //- L1 alla quota di carico
  //       TestALReady:=FALSE;
  //       IF ABS(Axes[L1].PosAx.positioningState.actualPosition-Programmi[ProgrammaAttivo].DatiAL.L1PosCarico)<pm[L1].ma_standstill_pos_tol THEN
  //         IF i_sys_SenzaTubo=TRUE THEN
  //           TestALReady:=TRUE;
  //         ELSE
  //           IF readdigitalinput(NumInput:=INP_AL5_PINZA_APERTA_DX)=FALSE AND
  //              readdigitalinput(NumInput:=INP_AL5_PINZA_APERTA_SX)=FALSE THEN
  //             TestALReady:=TRUE;
  //           END_IF;
  //         END_IF;
  //       END_IF;
  //   END_CASE;
  // {
  // #endif  //Fine No MS0017
  // }
END_FUNCTION
// {
// #endif  //Fine AL_BLM
// }

FUNCTION AL5FrenoSollevatore

  VAR_EXTERNAL CONSTANT
    OUT_AL5_FRENO_FASCIO                          :INT;
  END_VAR

  VAR_INPUT
    Stato  :BOOL;
  END_VAR
  ;
  // {
  // #ifdef AL_BLM
  // }
    WriteDigitalOutput(NumOutput:=OUT_AL5_FRENO_FASCIO, Value:=Stato);
  // {
  // #endif  //Fine AL_BLM
  // }
END_FUNCTION

/**********************************
 * LOAD RESERVATION LIGHT SETTING *
 **********************************/
FUNCTION AL5LucePrenotazioneCarico

  VAR_EXTERNAL CONSTANT
    OUT_AL5_RICHIESTA_CARICO_FASCIO               :INT;
  END_VAR

  VAR_INPUT
    Stato  :BOOL;
  END_VAR
  // {
  // #ifdef AL_BLM
  // }
    WriteDigitalOutput(NumOutput:=OUT_AL5_RICHIESTA_CARICO_FASCIO, Value:=Stato);
  // {
  // #endif  //Fine AL_BLM
  // }
  ;
END_FUNCTION

/********************************************************************************
 * SETTING THE ^OUTPUT ENABLING THE LOADING ROBOT TO TAKE THE HOSE FROM THE ^AL *
 ********************************************************************************/
// {
// #ifdef AL_BLM
// }
  FUNCTION ALRobotProntoScarico

    VAR_EXTERNAL
      i_sys_DpCoupler                 :BOOL;
      i_sys_PnCoupler                 :BOOL;
      OAddress                        : ARRAY [0..MAXDIGITALOUTPUT] OF Digital_Output;
    END_VAR

    VAR_EXTERNAL CONSTANT
      MAXDIGITALOUTPUT                              :INT;
      OUT_CARICO_TUBO_PRESENTE_AL                   :INT;
      OUT_CARICO_TUBO_PRESENTE_AL_DPCOUPLER         :INT;
    END_VAR

    VAR_INPUT
      Stato      :BOOL;
      Programma  :INT;
    END_VAR
    VAR
      Uscita    :INT;
    END_VAR
    IF TestRobotDaAl(Programma:=Programma)=TRUE THEN
      IF (i_sys_DpCoupler=TRUE OR i_sys_PnCoupler=TRUE) AND
         oaddress[OUT_CARICO_TUBO_PRESENTE_AL].port=-1 AND
         oaddress[OUT_CARICO_TUBO_PRESENTE_AL].bit=-1 THEN
        Uscita:=OUT_CARICO_TUBO_PRESENTE_AL_DPCOUPLER;
      ELSE
        Uscita:=OUT_CARICO_TUBO_PRESENTE_AL;
      END_IF;
      WriteDigitalOutput(NumOutput:=Uscita, Value:=Stato, Verifica:=TRUE);
    END_IF;
  END_FUNCTION

/************************************************************************************
 * OUTLET SETTING THAT ENABLES THE LOADING ROBOT TO EVACUATE THE TUBE FROM THE^AL42 *
 ************************************************************************************/
  FUNCTION ALRobotTuboLibero

    VAR_EXTERNAL
      i_sys_DpCoupler                 :BOOL;
      i_sys_PnCoupler                 :BOOL;
      OAddress                        : ARRAY [0..MAXDIGITALOUTPUT] OF Digital_Output;
    END_VAR

    VAR_EXTERNAL CONSTANT
      MAXDIGITALOUTPUT                    :INT;

      OUT_CARICO_TUBO_LIBERO_AL                     :INT;
      OUT_CARICO_TUBO_LIBERO_AL_DPCOUPLER           :INT;
    END_VAR

    VAR_INPUT
      Stato      :BOOL;
      Programma :INT;
    END_VAR
    VAR
      Uscita    :INT;
    END_VAR
    IF TestRobotDaAl(Programma:=Programma)=TRUE THEN
      IF (i_sys_DpCoupler=TRUE OR i_sys_PnCoupler=TRUE) AND
         oaddress[OUT_CARICO_TUBO_LIBERO_AL].port=-1 AND
         oaddress[OUT_CARICO_TUBO_LIBERO_AL].bit=-1 THEN
        Uscita:=OUT_CARICO_TUBO_LIBERO_AL_DPCOUPLER;
      ELSE
        Uscita:=OUT_CARICO_TUBO_LIBERO_AL;
      END_IF;
      WriteDigitalOutput(NumOutput:=Uscita, Value:=Stato, Verifica:=TRUE);
    END_IF;
  END_FUNCTION

/****************************************************************
 * TRUE IF THE TWO SYNCHRONISATION SENSORS HAVE THE SAME STATUS *
 ****************************************************************/

FUNCTION TestSincrCatene:BOOL

  VAR_EXTERNAL
    TimerSystem                     :ARRAY[0..MAX_TIMER_SYSTEM-1] OF Timer;
  END_VAR

  VAR_EXTERNAL CONSTANT
    INP_AL5_SINCR_CATENA_SX                         :INT;
    INP_AL5_SINCR_CATENA_DX                         :INT;
    T_SINCR_CATENE_AL5	                            :INT;
    MAX_TIMER_SYSTEM 	                              :USINT;
  END_VAR

  VAR
    dret  :DINT;
  END_VAR
  ;
  // {
  // #ifdef AL_BLM
  // }
    IF TimerSystem[T_SINCR_CATENE_AL5].Value=0 THEN
      //Serve per inibite la verifica del sincronismo fin tanto che il timer non si è azzerato.
      IF (ReadDigitalInput(NumInput:=INP_AL5_SINCR_CATENA_SX, Verifica:=FALSE)=TRUE AND
          ReadDigitalInput(NumInput:=INP_AL5_SINCR_CATENA_DX, Verifica:=FALSE)=TRUE) OR
         (ReadDigitalInput(NumInput:=INP_AL5_SINCR_CATENA_SX, Verifica:=FALSE)=FALSE AND
          ReadDigitalInput(NumInput:=INP_AL5_SINCR_CATENA_DX, Verifica:=FALSE)=FALSE) THEN
          TestSincrCatene:=TRUE;
      ELSE
        TestSincrCatene:=FALSE;
      END_IF;
    ELSE
      TestSincrCatene:=TRUE;
    END_IF;
  // {
  // #endif
  // }
END_FUNCTION

/********************************************************************************************************
 * CHECK WHETHER A ROBOT LOAD THAT PICKS UP THE PART FROM THE^AL IS FORESEEN IN THE INDICATED PROGRAMME *
 ********************************************************************************************************/

FUNCTION TestRobotDaAL:BOOL

  VAR_EXTERNAL
    Programmi                      :ARRAY[0.._CONST_VAR_DEF._MPROGRAMS#MAXPROGRAMS - UINT#1] OF Programma;
  END_VAR

  VAR_EXTERNAL CONSTANT
    CARICO_AL_BLM_ROBOT                	            :SINT;
  END_VAR

  VAR_INPUT
    Programma  :DINT;
  END_VAR
  TestRobotDaAL:=programmi[Programma].TipoCarico=CARICO_AL_BLM_ROBOT;
END_FUNCTION

FUNCTION_BLOCK FB_Wait_disp

  VAR_EXTERNAL
    Disp                            :ARRAY[(FIRST_DEVICE)..(FIRST_DEVICE+_MAXDEVICES#MAXDEVICES-1)] OF Device;
    StatusTrace                     :BOOL;
    i_sys_OPMODE                    : INT;
  END_VAR

  VAR_EXTERNAL CONSTANT
    FIRST_DEVICE                    :INT;
    AUTOMODE                        :INT;
    TRC_DISPOSITIVI                 :INT;
  END_VAR

  VAR_INPUT
    Device			:INT;
    State				:INT;
    Trace				:BOOL:=TRUE;
  END_VAR
  VAR
    dret				:DINT;
    Attivazione	:BOOL;

		CURRENT_STATE	:INT:=GENERAL_STATE#STATE_INIT;
  END_VAR
	VAR_OUTPUT
		OutputState		:INT;
	END_VAR
	CASE CURRENT_STATE OF
		GENERAL_STATE#STATE_INIT:
			IF Disp[Device].Enable=TRUE THEN
				IF i_sys_OPMODE=AUTOMODE THEN
					//Serve per evitare di segnalare macchna ferma quando si attende un dispositivo complesso
					//la cui gestione dei tempi non è prevista da VGP
					Attivazione:=TRUE;
					StatusTrace:=TRUE;
				ELSE
					Attivazione:=FALSE;
				END_IF;
				CURRENT_STATE:=_FB_WaitDisp#STATE_ATTESA_DISPOSITIVO;
			ELSE
				CURRENT_STATE:=GENERAL_STATE#STATE_END;
			END_IF;

    _FB_WaitDisp#STATE_ATTESA_DISPOSITIVO:
			IF Disp[Device].Stato<>State OR Disp[Device].consenso_minus=FALSE OR Disp[Device].consenso_plus=FALSE THEN
				IF Trace=TRUE THEN
					Set_Trace(Code:=TRC_DISPOSITIVI+Device, Axis:=Device);
				END_IF;
			ELSE
				IF Attivazione=TRUE THEN
					StatusTrace:=FALSE;
				END_IF;
				IF Trace=TRUE THEN
					reset_trace(TRC_DISPOSITIVI+Device);
				END_IF;
				IF Disp[Device].SpegnimentoUscita=TRUE THEN
					IF Disp[Device].Stato=State THEN
						IF State=Disp[Device].limite_lavoro THEN
							WriteDigitalOutput(NumOutput:=Disp[Device].out_lavoro, Value:=FALSE);
						ELSE
							IF State=Disp[Device].limite_riposo THEN
								WriteDigitalOutput(NumOutput:=Disp[Device].out_riposo, Value:=FALSE);
							END_IF;
						END_IF;
					END_IF;
				END_IF;
				CURRENT_STATE:=GENERAL_STATE#STATE_END;
			END_IF;

		GENERAL_STATE#STATE_END:
			CURRENT_STATE:=GENERAL_STATE#STATE_INIT;
	END_CASE;
	OutputState:=CURRENT_STATE;
END_FUNCTION_BLOCK

FUNCTION_BLOCK FB_VerificaStop

  VAR_EXTERNAL CONSTANT
    i_sys_stopcond                          : INT;
  END_VAR

  VAR
		CURRENT_STATE:INT:=GENERAL_STATE#STATE_INIT;
  END_VAR
	VAR_OUTPUT
		OutputState	:INT:=GENERAL_STATE#STATE_INIT;
	END_VAR
	CASE CURRENT_STATE OF
		GENERAL_STATE#STATE_INIT:
			IF NOT (i_sys_StopCond=1) THEN
				CURRENT_STATE:=GENERAL_STATE#STATE_END;
			END_IF;

		GENERAL_STATE#STATE_END:
			CURRENT_STATE:=GENERAL_STATE#STATE_INIT;
	END_CASE;
	OutputState:=CURRENT_STATE;
END_FUNCTION_BLOCK

/*************************************************************
 * SETS THE DIGITAL OUTPUTS FOR SELECTING THE PROTECTED AREA *
 *************************************************************/
FUNCTION AttivaProgrammaRadar

  VAR_EXTERNAL CONSTANT
    OUT_RADAR_0                                 :INT; //Gestione RADAR
    OUT_RADAR_1                                 :INT; //Gestione RADAR
    OUT_RADAR_2                                 :INT; //Gestione RADAR
    OUT_RADAR_3                                 :INT; //Gestione RADAR
  END_VAR

  VAR_INPUT
    Codice:  INT;
  END_VAR
  // {
  // #ifdef PROFINET
  // }
    // {
    // #ifndef RUNNER %%%%
    // }
    //   {
    //   #ifndef EFLEX_DH4010
    //   }
    //     CASE Codice OF
    //       0:O_Radar_Zona_1:=FALSE;
    //         O_Radar_Zona_2:=FALSE;
    //         O_Radar_Zona_3:=FALSE;
    //       1:O_Radar_Zona_1:=TRUE;
    //         O_Radar_Zona_2:=FALSE;
    //         O_Radar_Zona_3:=FALSE;
    //       2:O_Radar_Zona_1:=FALSE;
    //         O_Radar_Zona_2:=TRUE;
    //         O_Radar_Zona_3:=FALSE;
    //       3:O_Radar_Zona_1:=FALSE;
    //         O_Radar_Zona_2:=FALSE;
    //         O_Radar_Zona_3:=TRUE;
    //     END_CASE;
    //   {
    //   #endif  //FINE NO EFLEX_DH4010
    //   }
    // {
    // #endif  //Fine NO RUNNER
    // }
  // {
  // #else  //Fine PROFINET
  // }
    CASE Codice OF
      1:WriteDigitalOutput(NumOutput:=OUT_RADAR_0, Value:=BOOL#0, Verifica:=TRUE);
        WriteDigitalOutput(NumOutput:=OUT_RADAR_1, Value:=BOOL#1, Verifica:=TRUE);
        WriteDigitalOutput(NumOutput:=OUT_RADAR_2, Value:=BOOL#0, Verifica:=TRUE);
        WriteDigitalOutput(NumOutput:=OUT_RADAR_3, Value:=BOOL#0, Verifica:=TRUE);

      2:WriteDigitalOutput(NumOutput:=OUT_RADAR_0, Value:=BOOL#1, Verifica:=TRUE);
        WriteDigitalOutput(NumOutput:=OUT_RADAR_1, Value:=BOOL#0, Verifica:=TRUE);
        WriteDigitalOutput(NumOutput:=OUT_RADAR_2, Value:=BOOL#0, Verifica:=TRUE);
        WriteDigitalOutput(NumOutput:=OUT_RADAR_3, Value:=BOOL#0, Verifica:=TRUE);

      3:WriteDigitalOutput(NumOutput:=OUT_RADAR_0, Value:=BOOL#0, Verifica:=TRUE);
        WriteDigitalOutput(NumOutput:=OUT_RADAR_1, Value:=BOOL#0, Verifica:=TRUE);
        WriteDigitalOutput(NumOutput:=OUT_RADAR_2, Value:=BOOL#0, Verifica:=TRUE);
        WriteDigitalOutput(NumOutput:=OUT_RADAR_3, Value:=BOOL#1, Verifica:=TRUE);
    END_CASE;
  // {
  // #endif    //Fine NO PROFINET
  // }
  ;
END_FUNCTION

FUNCTION ResetCodificaPezzo
  // {
  // #ifdef CARICO_AUTOMATICO %%%%
  // }
	// 	WriteDigitalOutput(NumOutput:=OUT_SELEZ_PEZZO_BIT0, Value:=FALSE, Verifica:=FALSE);
	// 	WriteDigitalOutput(NumOutput:=OUT_SELEZ_PEZZO_BIT1, Value:=FALSE, Verifica:=FALSE);
	// 	WriteDigitalOutput(NumOutput:=OUT_SELEZ_PEZZO_BIT2, Value:=FALSE, Verifica:=FALSE);
	// 	WriteDigitalOutput(NumOutput:=OUT_SELEZ_PEZZO_BIT3, Value:=FALSE, Verifica:=FALSE);
	// 	WriteDigitalOutput(NumOutput:=OUT_SELEZ_PEZZO_BIT4, Value:=FALSE, Verifica:=FALSE);
	// 	WriteDigitalOutput(NumOutput:=OUT_SELEZ_PEZZO_BIT5, Value:=FALSE, Verifica:=FALSE);
	// 	WriteDigitalOutput(NumOutput:=OUT_SELEZ_PEZZO_BIT6, Value:=FALSE, Verifica:=FALSE);
	// 	WriteDigitalOutput(NumOutput:=OUT_PEZZO_ESEGUITO_BIT0_DPCOUPLER, Value:=FALSE, Verifica:=FALSE);
	// 	WriteDigitalOutput(NumOutput:=OUT_PEZZO_ESEGUITO_BIT1_DPCOUPLER, Value:=FALSE, Verifica:=FALSE);
	// 	WriteDigitalOutput(NumOutput:=OUT_PEZZO_ESEGUITO_BIT2_DPCOUPLER, Value:=FALSE, Verifica:=FALSE);
	// 	WriteDigitalOutput(NumOutput:=OUT_PEZZO_ESEGUITO_BIT3_DPCOUPLER, Value:=FALSE, Verifica:=FALSE);
	// 	WriteDigitalOutput(NumOutput:=OUT_PEZZO_ESEGUITO_BIT4_DPCOUPLER, Value:=FALSE, Verifica:=FALSE);
	// 	WriteDigitalOutput(NumOutput:=OUT_PEZZO_ESEGUITO_BIT5_DPCOUPLER, Value:=FALSE, Verifica:=FALSE);
	// 	WriteDigitalOutput(NumOutput:=OUT_PEZZO_ESEGUITO_BIT6_DPCOUPLER, Value:=FALSE, Verifica:=FALSE);
	// 	{
	// 	#ifdef PROFINET
	// 	}
	// 		pncoupler_o51:=0;
	// 	{
	// 	#endif  //Fine PROFINET
	// 	}
	// 	dbcoupler_o51:=0;
	// {
  // #endif  //Fine CARICO_AUTOMATICO
  // }
  ;
END_FUNCTION

/*******************************************************************************
 * SETTING ON X1 AXIS WITH ABSOLUTE ENCODER, OF THE OFFSET CALCULATED BY VGP3D *
 *******************************************************************************/

FUNCTION ImpostazioneOffsetX1
  VAR_INPUT
    Offset:LREAL;
  END_VAR
  VAR
    dret  :DINT;
    Delta  :LREAL;
  END_VAR
  // {
  // #ifndef ORBITALE
  // }
  //   IF pm[X1].ma_num_encs=1 THEN
  //     Delta:=Assi[X1].PosAx.positioningstate.actualposition-Assi[X1].PosAx.sensordata[1].position;
  //     IF ABS(Offset-Delta)>0.1 THEN
  //       dret:=_redefineposition(axis:=Assi[X1].PosAx,
  //                               redefinespecification:=COMMAND_VALUE,
  //                               redefinemode:=RELATIVE,
  //                               position:=Offset-Delta,
  //                               nextcommand:=WHEN_COMMAND_DONE);
  //     END_IF;
  //   END_IF;
  // {
  // #endif  //Fine NO ORBITALE
  // }
  ;
END_FUNCTION

//Verifica se l^asse passato come parametro è un bloccaggio
FUNCTION TestAsseBloccaggio:BOOL

  VAR_EXTERNAL CONSTANT
    W3 :    INT;
  END_VAR

  VAR_INPUT
    Asse  :INT;
  END_VAR;
  // {
  // #ifdef BLOCCAGGIO_SX %%%%
  // }
  //   TestAsseBloccaggio:=(Asse=W3) OR (Asse=W5);
  // {
  // #else    //Fine BLOCCAGGIO_SX
  // }
    // {
    // #ifdef BLOCCAGGIO_DX
    // }
      TestAsseBloccaggio:=(Asse=W3);
    // {
    // #endif    //Fine BLOCCAGGIO_DX
    // }
  // {
  // #endif    //Fine NO BLOCCAGGIO_SX
  // }
END_FUNCTION

/*************************************************************************
 * SETS THE ^ ACTIVE TOOL TO INDEFINITE IF ONE OF THE HEAD AXES IS MOVED *
 *************************************************************************/
FUNCTION TestAsseUtensile
  VAR_INPUT
    Asse  :INT;
  END_VAR
  // {
  // #ifdef CURVATURA
  // }
  //   {
  //   #ifdef EFLEX_DH4010
  //   }
  //     {
  //     #ifdef EFLEX
  //     }
  //       IF Asse=Q1 THEN
  //         i_sys_utensileAttivo:=0;
  //       END_IF;
  //     {
  //     #endif    //Fine EFLEX
  //     }
  //     {
  //     #ifdef DH4010
  //     }
  //       CASE Asse OF
  //         Q1:i_sys_utensileAttivo[TABELLA_SX]:=0;
  //         Q2:i_sys_utensileAttivo[TABELLA_DX]:=0;
  //       END_CASE
  //     {
  //     #endif    //Fine DH4010
  //     }
  //   {
  //   #else    //Fine EFLEX_DH4010
  //   }
  //     IF Asse=V1 OR Asse=Q1 THEN
  //       i_sys_utensileAttivo:=0;
  //     END_IF;
  //   {
  //   #endif  //Fine NO EFLEX_DH4010
  //   }
  // {
  // #endif  //Fine CURVATURA
  // }
  ;
END_FUNCTION

/***********************************************
 * READS THE ACTIVE SAFETY STATUS ON THE^DRIVE *
 ***********************************************/

// {
// ::ifdef PROFINET
// }
  FUNCTION ReadStateSafety:DWORD

    VAR_EXTERNAL
      StatoSafetety_X1:WORD;
      StatoSafetety_Y1:WORD;
      StatoSafetety_Z1:WORD;
      StatoSafetety_Q1:WORD;
      StatoSafetety_R1:WORD;
      StatoSafetety_W3:WORD;
      StatoSafetety_W4:WORD;
      StatoSafetety_U4:WORD;
      StatoSafetety_L1:WORD;
      StatoSafetety_Z2:WORD;
    END_VAR

    VAR_EXTERNAL CONSTANT
      Z2  :INT;
      X1:INT;

      Y1:INT;

      Z1:INT;

      Q1:INT;

      V1:INT;
      W3 : INT;
      W4 :INT;
      U4 :INT;
      L1 :INT;

    END_VAR

    VAR_INPUT
      Asse  :INT;
    END_VAR
    ;
    // {
    // #ifndef EMULAZIONE
    // }
      // {
      // #ifdef ORBITALE
      // }
      //   CASE Asse OF
      //     {
      //     #ifdef RUNNER
      //     }
      //       X1:
      //         ReadStateSafety:=StatoSafetety_X1;
      //       W2:
      //         ReadStateSafety:=StatoSafetety_W2;
      //       U1:
      //         ReadStateSafety:=StatoSafetety_U1;
      //       U2:
      //         ReadStateSafety:=StatoSafetety_U2;
      //       {
      //       #ifndef PLAUNO_LIGHT
      //       }
      //         W1:
      //           ReadStateSafety:=StatoSafetety_W1;
      //         A1:
      //           ReadStateSafety:=StatoSafetety_A1;
      //         {
      //         #ifndef THREE_RUNNER
      //         }
      //           A2:
      //             ReadStateSafety:=StatoSafetety_A2;
      //         {
      //         #endif //FINE NO THREE_RUNNER
      //         }
      //       {
      //       #endif //FINE NO PLAUNO_LIGHT
      //       }
      //       {
      //       #ifdef FOUR_RUNNER_PLAUNO
      //       }
      //         Y1:
      //           ReadStateSafety:=StatoSafetety_Y1;
      //         Z1:
      //           ReadStateSafety:=StatoSafetety_Z1;
      //         Q1:
      //           ReadStateSafety:=StatoSafetety_Q1;
      //         V1:
      //           ReadStateSafety:=StatoSafetety_V1;
      //         W3:
      //           ReadStateSafety:=StatoSafetety_W3;
      //         {
      //         #ifdef SPALLAMENTO_DX
      //         }
      //           W4:
      //             ReadStateSafety:=StatoSafetety_W4;
      //         {
      //         #endif    //Fine SPALLAMENTO_DX
      //         }
      //         {
      //         #ifdef FOUR_RUNNER
      //         }
      //           V2:
      //             ReadStateSafety:=StatoSafetety_V2;
      //         {
      //         #endif    //Fine FOUR_RUNNER
      //         }

      //       {
      //       #endif    //Fine FOUR_RUNNER_PLAUNO
      //       }
      //       {
      //       #ifdef B1_B2
      //       }
      //         B1:
      //           ReadStateSafety:=StatoSafetety_B1;
      //         B2:
      //           ReadStateSafety:=StatoSafetety_B2;
      //       {
      //       #endif    //Fine B1_B2
      //       }
      //     {
      //     #endif    //Fine RUNNER
      //     }
      //     {
      //     #ifdef EFLEX
      //     }
      //                   X1:
      //                       ReadStateSafety:=StatoSafetety_X1;
      //                   Y1:
      //                       ReadStateSafety:=StatoSafetety_Y1;
      //                   Z1:
      //                       ReadStateSafety:=StatoSafetety_Z1;
      //                   Q1:
      //                       ReadStateSafety:=StatoSafetety_Q1;
      //       W1:
      //         ReadStateSafety:=StatoSafetety_W1;
      //     {
      //     #endif    //EFLEX
      //     }
      //     {
      //     #ifdef DH4010
      //     }
      //                   X1:
      //                       ReadStateSafety:=StatoSafetety_X1;
      //                   X2:
      //                       ReadStateSafety:=StatoSafetety_X2;
      //                   Y1:
      //                       ReadStateSafety:=StatoSafetety_Y1;
      //                   Y2:
      //                       ReadStateSafety:=StatoSafetety_Y2;
      //                   Q1:
      //                       ReadStateSafety:=StatoSafetety_Q1;
      //                   Q2:
      //                       ReadStateSafety:=StatoSafetety_Q2;
      //                   Z1:
      //                       ReadStateSafety:=StatoSafetety_Z1;
      //       X3:
      //         ReadStateSafety:=StatoSafetety_X3;
      //       X6:
      //         ReadStateSafety:=StatoSafetety_X6;
      //     {
      //     #endif    //DH4010
      //     }
      //   ELSE
      //     ReadStateSafety:=1;
      //   END_CASE;
      // {
      // #else    //Fine macchine oribitali
      // }
        CASE Asse OF
          X1:
            ReadStateSafety:=StatoSafetety_X1;
          Y1:
            ReadStateSafety:=StatoSafetety_Y1;
          Z1:
            ReadStateSafety:=StatoSafetety_Z1;
          Q1:
            ReadStateSafety:=StatoSafetety_Q1;
          V1:
            ReadStateSafety:=StatoSafetety_R1;
          // {
          // #ifdef BLOCCAGGIO_DX
          // }
                        W3:
                            ReadStateSafety:=StatoSafetety_W3;
          // {
          // #endif    //Fine BLOCCAGGIO_DX
          // }
          // {
          // #ifdef SPALLAMENTO_DX
          // }
                        W4:
                            ReadStateSafety:=StatoSafetety_W4;
          // {
          // #endif    //Fine SPALLAMENTO_DX
          // }
          // {
          // #ifdef SLITTA_MOBILE_DX
          // }
                        U4:
                            ReadStateSafety:=StatoSafetety_U4;
          // {
          // #endif    //Fine SLITTA_MOBILE_DX
          // }
          // {
          // #ifdef NO_ASSE_U2 %%%%
          // }
          //               U2:
          //                   //Non esiste l^azionamento U2 si prende l^informazione da un asse sicuramente presente
          //                   ReadStateSafety:=StatoSafetety_Y1;
          // {
          // #else    //Fine NO_ASSE_U2
          // }
          //               U2:
          //                   ReadStateSafety:=StatoSafetety_U2;
          // {
          // #endif    //Fine NO NO_ASSE_U2
          // }
          // {
          // #ifdef BLOCCAGGIO_SX %%%%
          // }
          //   W5:
          //     ReadStateSafety:=StatoSafetety_W5;
          // {
          // #endif    //Fine BLOCCAGGIO_SX
          // }
          // {
          // #ifdef SPALLAMENTO_SX
          // }
          //   W6:
          //     ReadStateSafety:=StatoSafetety_W6;
          // {
          // #endif    //Fine SPALLAMENTO_SX
          // }
          // {
          // #ifdef SLITTA_MOBILE_SX
          // }
          //   U5:
          //     ReadStateSafety:=StatoSafetety_U5;
          // {
          // #endif    //Fine SLITTA_MOBILE_SX
          // }
					// {
					// #ifdef MATRICE_ELETTRICA
					// }
          //   Y2:
          //     ReadStateSafety:=StatoSafetety_Y2;
          // {
          // #endif    //Fine MATRICE_ELETTRICA
          // }
					// {
					// #ifdef SOLLEVAMENTO_SLITTA_SPALLAMENTO
					// }
          //   V4:
          //     ReadStateSafety:=StatoSafetety_V4;
					// {
					// #endif    //Fine SOLLEVAMENTO_SLITTA_SPALLAMENTO
					// }
          // {
          // #ifdef AL_BLM
          // }
            L1:
              ReadStateSafety:=StatoSafetety_L1;
          // {
          // #endif    //Fine AL_BLM
          // }
					// {
					// #ifdef ASSE_Z2
					// }
            Z2:
              ReadStateSafety:=StatoSafetety_Z2;
					// {
					// #endif //Fine ASSE_Z2
					// }
					// {
					// #ifdef PINZA_ELETTRICA
					// }
					// 	W1:
					// 		ReadStateSafety:=StatoSafetety_W1;
					// {
					// #endif //Fine PINZA_ELETTRICA
					// }
					// {
					// #ifdef SOSTEGNO_ELETTRICO
					// }
					// 	S1:
					// 		ReadStateSafety:=StatoSafetety_S1;
					// {
					// #endif //Fine SOSTEGNO_ELETTRICO
					// }
					// {
					// #ifdef BASCULANTE_ELETTRICO
					// }
					// 	B2:
					// 		ReadStateSafety:=StatoSafetety_B2;
					// {
					// #endif //Fine BASCULANTE_ELETTRICO
					// }
        ELSE
          ReadStateSafety:=DWORD#1;
        END_CASE;
      // {
      // #endif    //Fine NO ORBITALE
      // }
    // {
    // ::endif    //Fine NO EMULAZIONE
    // };
  END_FUNCTION
// {
// ::endif    //Fine PROFINET
// };

/***************************************************************
 * CHECKS WHETHER THE^AXIS PASSED AS A PARAMETER IS A SHOULDER *
 ***************************************************************/
FUNCTION TestAsseSpallamento:BOOL

  VAR_EXTERNAL CONSTANT
    W4:INT;
  END_VAR

  VAR_INPUT
    Asse  :INT;
  END_VAR;
    TestAsseSpallamento:=FALSE;
  // {
  // #ifdef SPALLAMENTO_SX
  // }
  //   TestAsseSpallamento:=(Asse=W4) OR (Asse=W6);
  // {
  // #else    //Fine SPALLAMENTO_SX
  // }
  {::ifdef SPALLAMENTO_DX}
      TestAsseSpallamento:=(Asse=W4);
  {::endif}    //Fine SPALLAMENTO_DX

END_FUNCTION

END_NAMESPACE
